// SIMATIC STEP 7 (V5.x) project COB2-CORDNT_040112_LATST
// CPU: CPU 315-2 DP
// station: Hardware
// station: SIMATIC 300(1)
// station: P_ADR_BUS
// program: S7 Program(1)

SYMBOL_TABLE
"DB:RxDTFrmPushCurrent"	DB 15	DB 15	// Pusher Current Data
"DB:RxDTFrmLavelleCurrent"	DB 16	DB 16
"DB: RxEDFrmCharger"	DB 17	DB 17
"DB: RxEDFrmGide"	DB 18	DB 18
"DB: RxEDFrmLoco"	DB 19	DB 19
"DB: RxEDFrmPusher"	DB 20	DB 20
"DB:TxDTFrmCo-Ordination"	DB 21	DB 21
"Level#1<< ---->>Level#2"	DB 23	DB 23
"DB:Data_ReciveBuffer"	DB 29	DB 29
"DB: AutoSPOT"	DB 31	DB 31
"DB: RFModem Freq"	DB 32	DB 32
"DB:HMI TagList"	DB 35	DB 35
"DB:User"	DB 36	DB 36
"DB:InitializationRxBuffe"	DB 39	DB 39
"DB:SndWork DB RS232C"	DB 40	DB 40	// Work DB for P_SND_RK
"DB:RevWork DB RS232C"	DB 41	DB 41	// Work DB for P_RCV_RK
"testng_4_ram_curent_fc45"	DB 45	DB 45	// testng_4_ram_curent_fc45
"FOR_FC-45-OFFLINE"	DB 46	DB 46	// FOR_FC-45-OFFLINE
"IDB_RS232_RM_ChgFreq_SND"	DB 50	FB 8
"IDB_RS232_RM_ChgFreq_RCV"	DB 51	FB 7
"IDB_RS485_AutoSPOT_RCV"	DB 80	FB 7
"DB:USE"	DB 100	DB 100
"P_RCV_ASCII"	FB 7	FB 7	// Receive Data / Provide Data
"P_SND_ASCII"	FB 8	FB 8	// Send Data / Fetch Data
"FC:RF CommunicaTion"	FC 14	FC 14	// RF--Communication & Data Handaling
"FC:OvenIdentification"	FC 19	FC 19
"FC:RxTeleGrm Alocation"	FC 20	FC 20
"FC:RFSndTGram"	FC 21	FC 21	// RF Telegram Sanding
"FC:TxSandTrigger"	FC 23	FC 23
"FC:Co-Ordination Process"	FC 24	FC 24
"FC:SCH_HandLing"	FC 25	FC 25
"FC:CoPLC-------->HMI"	FC 26	FC 26
"FC:FreqChanging"	FC 28	FC 28
"FC:RS232C RCV BLOCK"	FC 29	FC 29
"FC:RS232C SND BLOCK"	FC 30	FC 30	// Communications
"FC: RdAutoSPOT"	FC 31	FC 31	// Oven Identification
"FC:Group_Change_Info"	FC 40	FC 40
"FC_45_OFFLINE"	FC 45	FC 45	// FC_45_OFFLINE
"LoG_0"	M 0.0	BOOL	// LOG 0 BIT
"LoG_1"	M 0.1	BOOL	// LOG 1 BIT
"SysClk_1Sec"	M 1.5	BOOL
"SysClk_2Sec"	M 1.7	BOOL
"CYCL_EXC"	OB 1	OB 1	// Cycle Execution
"PROG_ERR"	OB 121	OB 121	// Programming Error
"MOD_ERR"	OB 122	OB 122	// Module Access Error
"RDREC"	SFB 52	SFB 52	// Read a Process Data Record
"WRREC"	SFB 53	SFB 53	// Write a Process Data Record
"BLKMOV"	SFC 20	SFC 20	// Copy Variables
"FILL"	SFC 21	SFC 21	// Initialize a Memory Area
"VAT_1"	VAT 1	
"ram current testing"	VAT 2		// ram current testing
"all car pos"	VAT 3		// all car pos
"VAT_4"	VAT 4	
"vat5_for_schedule_chek"	VAT 5		// vat5_for_schedule_chek
END_SYMBOL_TABLE

// FB 7: know-how protected block, not included

// FB 8: know-how protected block, not included

FUNCTION "FC:RF CommunicaTion" : VOID	// FC 14
VERSION : 0.1
BEGIN
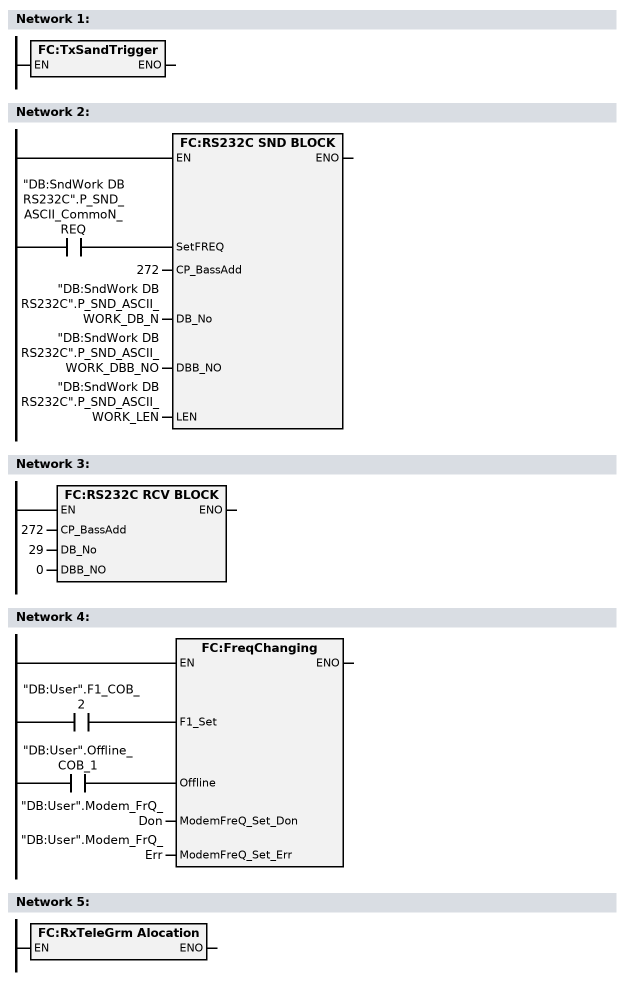
NETWORK
TITLE =
      CALL  "FC:TxSandTrigger";
      NOP   0;
NETWORK
TITLE =
//Data Sand Function Of Radio Modem
      A     "DB:SndWork DB RS232C".P_SND_ASCII_CommoN_REQ;
      =     L 0.0;
      BLD   103;
      CALL  "FC:RS232C SND BLOCK" (
           SetFREQ                  := L 0.0,
           CP_BassAdd               := 272,
           DB_No                    := "DB:SndWork DB RS232C".P_SND_ASCII_WORK_DB_N,
           DBB_NO                   := "DB:SndWork DB RS232C".P_SND_ASCII_WORK_DBB_NO,
           LEN                      := "DB:SndWork DB RS232C".P_SND_ASCII_WORK_LEN);
      NOP   0;
NETWORK
TITLE =
//Data Recive Function Of Radio Modem
      CALL  "FC:RS232C RCV BLOCK" (
           CP_BassAdd               := 272,
           DB_No                    := 29,
           DBB_NO                   := 0);
      NOP   0;
NETWORK
TITLE =
//RF-- Frequency Set In Co-Ordination PLc
      A     "DB:User".F1_COB_2;
      =     L 0.0;
      BLD   103;
      A     "DB:User".Offline_COB_1;
      =     L 0.1;
      BLD   103;
      CALL  "FC:FreqChanging" (
           F1_Set                   := L 0.0,
           Offline                  := L 0.1,
           ModemFreQ_Set_Don        := "DB:User".Modem_FrQ_Don,
           ModemFreQ_Set_Err        := "DB:User".Modem_FrQ_Err);
      NOP   0;
NETWORK
TITLE =
      CALL  "FC:RxTeleGrm Alocation";
      NOP   0;
END_FUNCTION

FUNCTION "FC:OvenIdentification" : VOID	// FC 19
AUTHOR : SKD
NAME : CDSPL
VERSION : 0.1
BEGIN
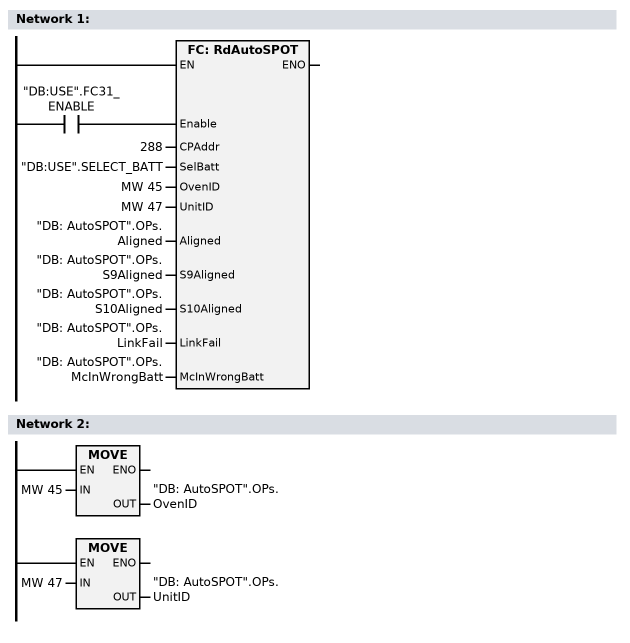
NETWORK
TITLE =
      A     "DB:USE".FC31_ENABLE;
      =     L 0.0;
      BLD   103;
      CALL  "FC: RdAutoSPOT" (
           Enable                   := L 0.0,
           CPAddr                   := 288,
           SelBatt                  := "DB:USE".SELECT_BATT,
           OvenID                   := MW 45,
           UnitID                   := MW 47,
           Aligned                  := "DB: AutoSPOT".OPs.Aligned,
           S9Aligned                := "DB: AutoSPOT".OPs.S9Aligned,
           S10Aligned               := "DB: AutoSPOT".OPs.S10Aligned,
           LinkFail                 := "DB: AutoSPOT".OPs.LinkFail,
           McInWrongBatt            := "DB: AutoSPOT".OPs.McInWrongBatt);
      NOP   0;
NETWORK
TITLE =
      L     MW 45;
      T     "DB: AutoSPOT".OPs.OvenID;
//..
      L     MW 47;
      T     "DB: AutoSPOT".OPs.UnitID;
END_FUNCTION

FUNCTION "FC:RxTeleGrm Alocation" : VOID	// FC 20
VERSION : 0.1
BEGIN
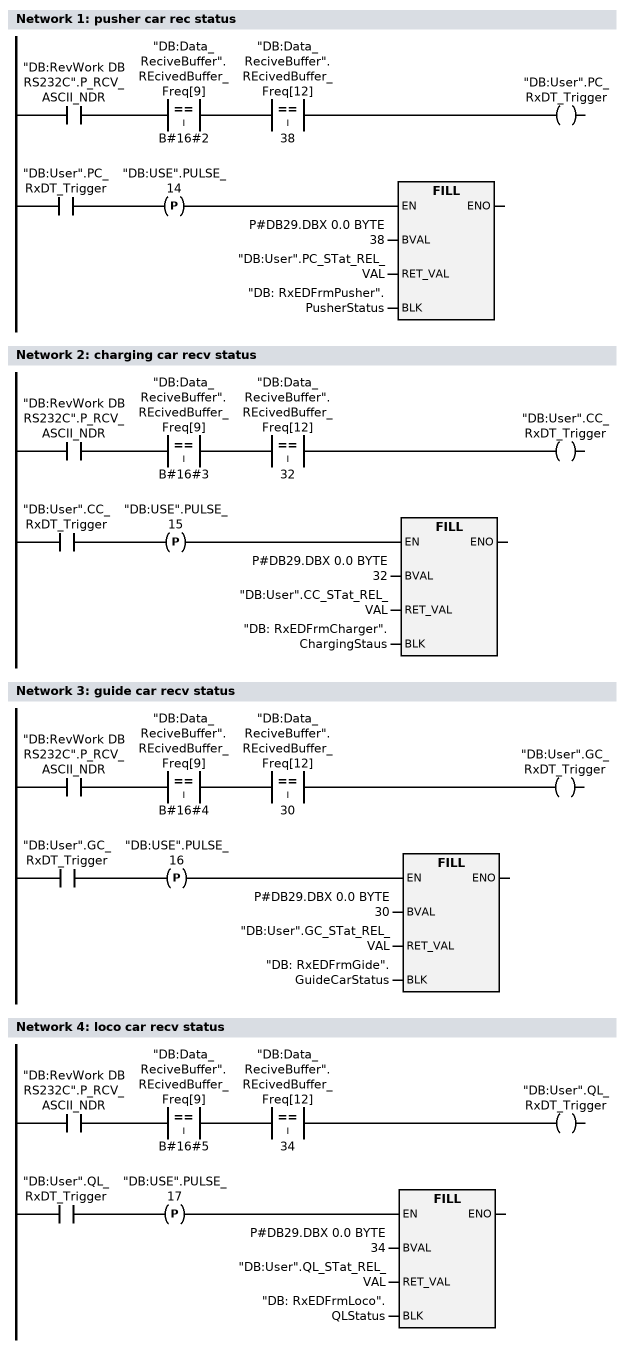
NETWORK
TITLE = pusher car rec status
//pusher car rec status
      A     "DB:RevWork DB RS232C".P_RCV_ASCII_NDR;
      A(;
      L     "DB:Data_ReciveBuffer".REcivedBuffer_Freq[9];
      L     B#16#2;
      ==I;
      );
      A(;
      L     "DB:Data_ReciveBuffer".REcivedBuffer_Freq[12];
      L     38;	//Massege ID
      ==I;
      );
      =     "DB:User".PC_RxDT_Trigger;
//..
      A     "DB:User".PC_RxDT_Trigger;
      FP    "DB:USE".PULSE_14;
      JNB   PC00;
      CALL  "FILL" (
           BVAL                     := P#DB29.DBX 0.0 BYTE 38,
           RET_VAL                  := "DB:User".PC_STat_REL_VAL,
           BLK                      := "DB: RxEDFrmPusher".PusherStatus);
PC00: NOP   0;
NETWORK
TITLE = charging car recv status
//charging car recv status
      A     "DB:RevWork DB RS232C".P_RCV_ASCII_NDR;
      A(;
      L     "DB:Data_ReciveBuffer".REcivedBuffer_Freq[9];
      L     B#16#3;
      ==I;
      );
      A(;
      L     "DB:Data_ReciveBuffer".REcivedBuffer_Freq[12];
      L     32;	//Massege ID
      ==I;
      );
      =     "DB:User".CC_RxDT_Trigger;
//..
      A     "DB:User".CC_RxDT_Trigger;
      FP    "DB:USE".PULSE_15;
      JNB   CC00;
      CALL  "FILL" (
           BVAL                     := P#DB29.DBX 0.0 BYTE 32,
           RET_VAL                  := "DB:User".CC_STat_REL_VAL,
           BLK                      := "DB: RxEDFrmCharger".ChargingStaus);
CC00: NOP   0;
NETWORK
TITLE = guide car recv status
//guide car recv status
      A     "DB:RevWork DB RS232C".P_RCV_ASCII_NDR;
      A(;
      L     "DB:Data_ReciveBuffer".REcivedBuffer_Freq[9];
      L     B#16#4;
      ==I;
      );
      A(;
      L     "DB:Data_ReciveBuffer".REcivedBuffer_Freq[12];
      L     30;	//Massege ID
      ==I;
      );
      =     "DB:User".GC_RxDT_Trigger;
//..
      A     "DB:User".GC_RxDT_Trigger;
      FP    "DB:USE".PULSE_16;
      JNB   GC00;
      CALL  "FILL" (
           BVAL                     := P#DB29.DBX 0.0 BYTE 30,
           RET_VAL                  := "DB:User".GC_STat_REL_VAL,
           BLK                      := "DB: RxEDFrmGide".GuideCarStatus);
GC00: NOP   0;
NETWORK
TITLE = loco car recv status
//Quenching Car Status
      A     "DB:RevWork DB RS232C".P_RCV_ASCII_NDR;
      A(;
      L     "DB:Data_ReciveBuffer".REcivedBuffer_Freq[9];
      L     B#16#5;
      ==I;
      );
      A(;
      L     "DB:Data_ReciveBuffer".REcivedBuffer_Freq[12];
      L     34;	//Massege ID
      ==I;
      );
      =     "DB:User".QL_RxDT_Trigger;
//..
      A     "DB:User".QL_RxDT_Trigger;
      FP    "DB:USE".PULSE_17;
      JNB   QL00;
      CALL  "FILL" (
           BVAL                     := P#DB29.DBX 0.0 BYTE 34,
           RET_VAL                  := "DB:User".QL_STat_REL_VAL,
           BLK                      := "DB: RxEDFrmLoco".QLStatus);
QL00: NOP   0;
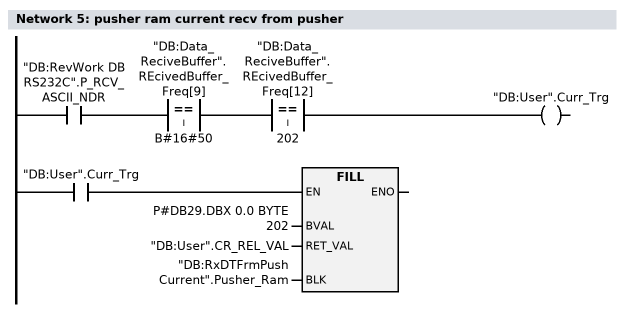
NETWORK
TITLE = pusher ram current recv from pusher
//pusher ram current recv from pusher
      A     "DB:RevWork DB RS232C".P_RCV_ASCII_NDR;
      A(;
      L     "DB:Data_ReciveBuffer".REcivedBuffer_Freq[9];
      L     B#16#50;
      ==I;
      );
      A(;
      L     "DB:Data_ReciveBuffer".REcivedBuffer_Freq[12];
      L     202;	//Massege ID
      ==I;
      );
      =     "DB:User".Curr_Trg;
//..
      A     "DB:User".Curr_Trg;
      JNB   CR00;
      CALL  "FILL" (
           BVAL                     := P#DB29.DBX 0.0 BYTE 202,
           RET_VAL                  := "DB:User".CR_REL_VAL,
           BLK                      := "DB:RxDTFrmPushCurrent".Pusher_Ram);
CR00: NOP   0;
END_FUNCTION

FUNCTION "FC:RFSndTGram" : VOID	// FC 21
VERSION : 0.1
BEGIN
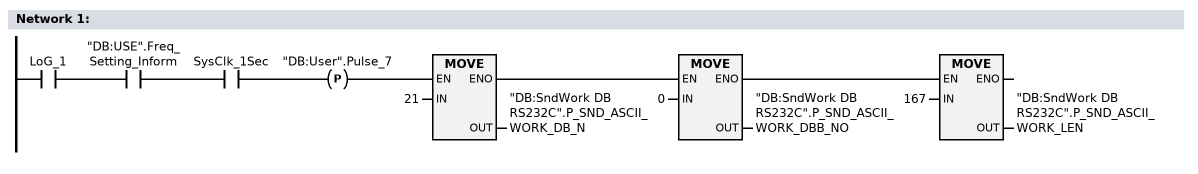
NETWORK
TITLE =
      A(;
      A(;
      A     "LoG_1";
      A     "DB:USE".Freq_Setting_Inform;
      A     "SysClk_1Sec";
      FP    "DB:User".Pulse_7;
      JNB   _001;
      L     21;
      T     "DB:SndWork DB RS232C".P_SND_ASCII_WORK_DB_N;
      SET;
      SAVE;
      CLR;
_001: A     BR;
      );
      JNB   _002;
      L     0;
      T     "DB:SndWork DB RS232C".P_SND_ASCII_WORK_DBB_NO;
      SET;
      SAVE;
      CLR;
_002: A     BR;
      );
      JNB   _003;
      L     167;
      T     "DB:SndWork DB RS232C".P_SND_ASCII_WORK_LEN;
_003: NOP   0;
END_FUNCTION

FUNCTION "FC:TxSandTrigger" : VOID	// FC 23
VERSION : 0.1
BEGIN
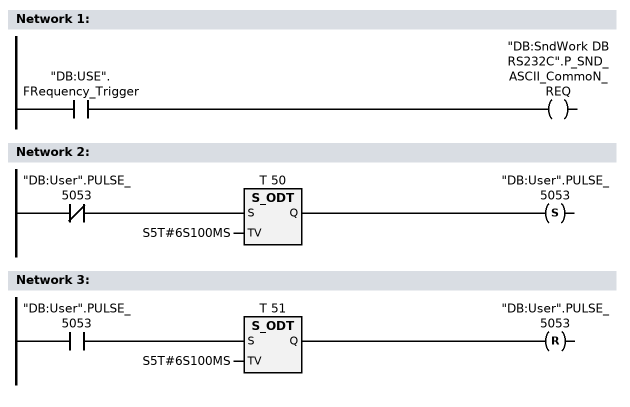
NETWORK
TITLE =
//Machine Grouping and Frequency Setting Triger....for Charging car
      A     "DB:USE".FRequency_Trigger;
      =     "DB:SndWork DB RS232C".P_SND_ASCII_CommoN_REQ;
NETWORK
TITLE =
      AN    "DB:User".PULSE_5053;
      L     S5T#6S100MS;
      SD    T 50;
      NOP   0;
      NOP   0;
      NOP   0;
      A     T 50;
      S     "DB:User".PULSE_5053;
NETWORK
TITLE =
      A     "DB:User".PULSE_5053;
      L     S5T#6S100MS;
      SD    T 51;
      NOP   0;
      NOP   0;
      NOP   0;
      A     T 51;
      R     "DB:User".PULSE_5053;
END_FUNCTION

FUNCTION "FC:Co-Ordination Process" : VOID	// FC 24
VERSION : 0.1
BEGIN
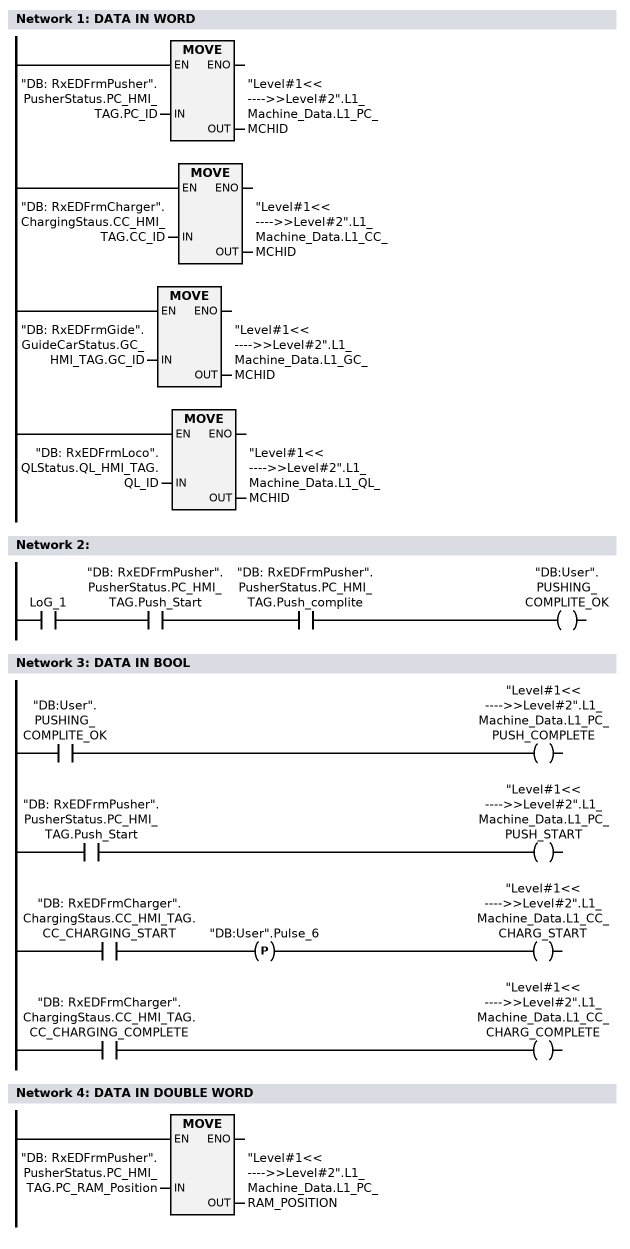
NETWORK
TITLE = DATA IN WORD
      L     "DB: RxEDFrmPusher".PusherStatus.PC_HMI_TAG.PC_ID;
      T     "Level#1<< ---->>Level#2".L1_Machine_Data.L1_PC_MCHID;
//..
      L     "DB: RxEDFrmCharger".ChargingStaus.CC_HMI_TAG.CC_ID;
      T     "Level#1<< ---->>Level#2".L1_Machine_Data.L1_CC_MCHID;
//..
      L     "DB: RxEDFrmGide".GuideCarStatus.GC_HMI_TAG.GC_ID;
      T     "Level#1<< ---->>Level#2".L1_Machine_Data.L1_GC_MCHID;
//..
      L     "DB: RxEDFrmLoco".QLStatus.QL_HMI_TAG.QL_ID;
      T     "Level#1<< ---->>Level#2".L1_Machine_Data.L1_QL_MCHID;
//...
NETWORK
TITLE =
      A     "LoG_1";
      A     "DB: RxEDFrmPusher".PusherStatus.PC_HMI_TAG.Push_Start;
      A     "DB: RxEDFrmPusher".PusherStatus.PC_HMI_TAG.Push_complite;
      =     "DB:User".PUSHING_COMPLITE_OK;
NETWORK
TITLE = DATA IN BOOL
      A     "DB:User".PUSHING_COMPLITE_OK;
      =     "Level#1<< ---->>Level#2".L1_Machine_Data.L1_PC_PUSH_COMPLETE;
//..
      A     "DB: RxEDFrmPusher".PusherStatus.PC_HMI_TAG.Push_Start;
      =     "Level#1<< ---->>Level#2".L1_Machine_Data.L1_PC_PUSH_START;
//..        
      A     "DB: RxEDFrmCharger".ChargingStaus.CC_HMI_TAG.CC_CHARGING_START;
      FP    "DB:User".Pulse_6;
      =     "Level#1<< ---->>Level#2".L1_Machine_Data.L1_CC_CHARG_START;
//..
      A     "DB: RxEDFrmCharger".ChargingStaus.CC_HMI_TAG.CC_CHARGING_COMPLETE;
      =     "Level#1<< ---->>Level#2".L1_Machine_Data.L1_CC_CHARG_COMPLETE;
NETWORK
TITLE = DATA IN DOUBLE WORD
      L     "DB: RxEDFrmPusher".PusherStatus.PC_HMI_TAG.PC_RAM_Position;
      T     "Level#1<< ---->>Level#2".L1_Machine_Data.L1_PC_RAM_POSITION;
//..
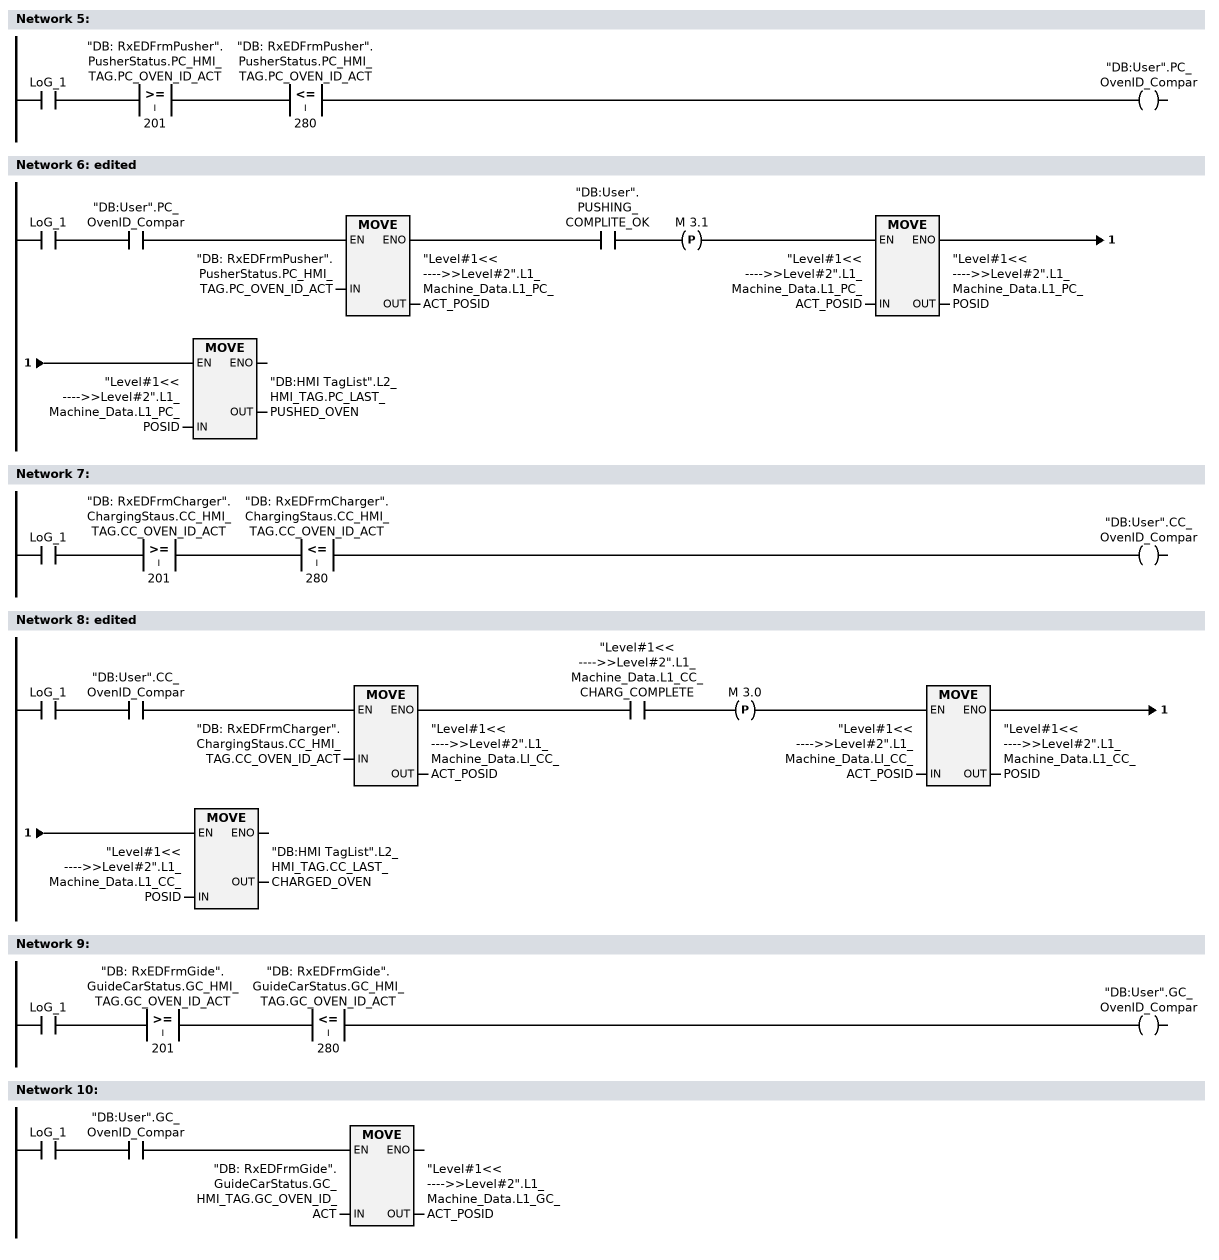
NETWORK
TITLE =
      A     "LoG_1";
      A(;
      L     "DB: RxEDFrmPusher".PusherStatus.PC_HMI_TAG.PC_OVEN_ID_ACT;
      L     201;
      >=I;
      );
      A(;
      L     "DB: RxEDFrmPusher".PusherStatus.PC_HMI_TAG.PC_OVEN_ID_ACT;
      L     280;
      <=I;
      );
      =     "DB:User".PC_OvenID_Compar;
NETWORK
TITLE = edited
//edited last 3  element in this n/w 8 & 6 by me for PC
      A(;
      A(;
      A     "LoG_1";
      A     "DB:User".PC_OvenID_Compar;
      JNB   _001;
      L     "DB: RxEDFrmPusher".PusherStatus.PC_HMI_TAG.PC_OVEN_ID_ACT;
      T     "Level#1<< ---->>Level#2".L1_Machine_Data.L1_PC_ACT_POSID;
      SET;
      SAVE;
      CLR;
_001: A     BR;
      );
      A     "DB:User".PUSHING_COMPLITE_OK;
      FP    M 3.1;
      JNB   _002;
      L     "Level#1<< ---->>Level#2".L1_Machine_Data.L1_PC_ACT_POSID;
      T     "Level#1<< ---->>Level#2".L1_Machine_Data.L1_PC_POSID;
      SET;
      SAVE;
      CLR;
_002: A     BR;
      );
      JNB   _003;
      L     "Level#1<< ---->>Level#2".L1_Machine_Data.L1_PC_POSID;
      T     "DB:HMI TagList".L2_HMI_TAG.PC_LAST_PUSHED_OVEN;
_003: NOP   0;
NETWORK
TITLE =
      A     "LoG_1";
      A(;
      L     "DB: RxEDFrmCharger".ChargingStaus.CC_HMI_TAG.CC_OVEN_ID_ACT;
      L     201;
      >=I;
      );
      A(;
      L     "DB: RxEDFrmCharger".ChargingStaus.CC_HMI_TAG.CC_OVEN_ID_ACT;
      L     280;
      <=I;
      );
      =     "DB:User".CC_OvenID_Compar;
NETWORK
TITLE = edited
//edited last 3  element in this n/w 8 & 6 by me for CC
      A(;
      A(;
      A     "LoG_1";
      A     "DB:User".CC_OvenID_Compar;
      JNB   _004;
      L     "DB: RxEDFrmCharger".ChargingStaus.CC_HMI_TAG.CC_OVEN_ID_ACT;
      T     "Level#1<< ---->>Level#2".L1_Machine_Data.LI_CC_ACT_POSID;
      SET;
      SAVE;
      CLR;
_004: A     BR;
      );
      A     "Level#1<< ---->>Level#2".L1_Machine_Data.L1_CC_CHARG_COMPLETE;
      FP    M 3.0;
      JNB   _005;
      L     "Level#1<< ---->>Level#2".L1_Machine_Data.LI_CC_ACT_POSID;
      T     "Level#1<< ---->>Level#2".L1_Machine_Data.L1_CC_POSID;
      SET;
      SAVE;
      CLR;
_005: A     BR;
      );
      JNB   _006;
      L     "Level#1<< ---->>Level#2".L1_Machine_Data.L1_CC_POSID;
      T     "DB:HMI TagList".L2_HMI_TAG.CC_LAST_CHARGED_OVEN;
_006: NOP   0;
NETWORK
TITLE =
      A     "LoG_1";
      A(;
      L     "DB: RxEDFrmGide".GuideCarStatus.GC_HMI_TAG.GC_OVEN_ID_ACT;
      L     201;
      >=I;
      );
      A(;
      L     "DB: RxEDFrmGide".GuideCarStatus.GC_HMI_TAG.GC_OVEN_ID_ACT;
      L     280;
      <=I;
      );
      =     "DB:User".GC_OvenID_Compar;
NETWORK
TITLE =
      A     "LoG_1";
      A     "DB:User".GC_OvenID_Compar;
      JNB   _007;
      L     "DB: RxEDFrmGide".GuideCarStatus.GC_HMI_TAG.GC_OVEN_ID_ACT;
      T     "Level#1<< ---->>Level#2".L1_Machine_Data.L1_GC_ACT_POSID;
_007: NOP   0;
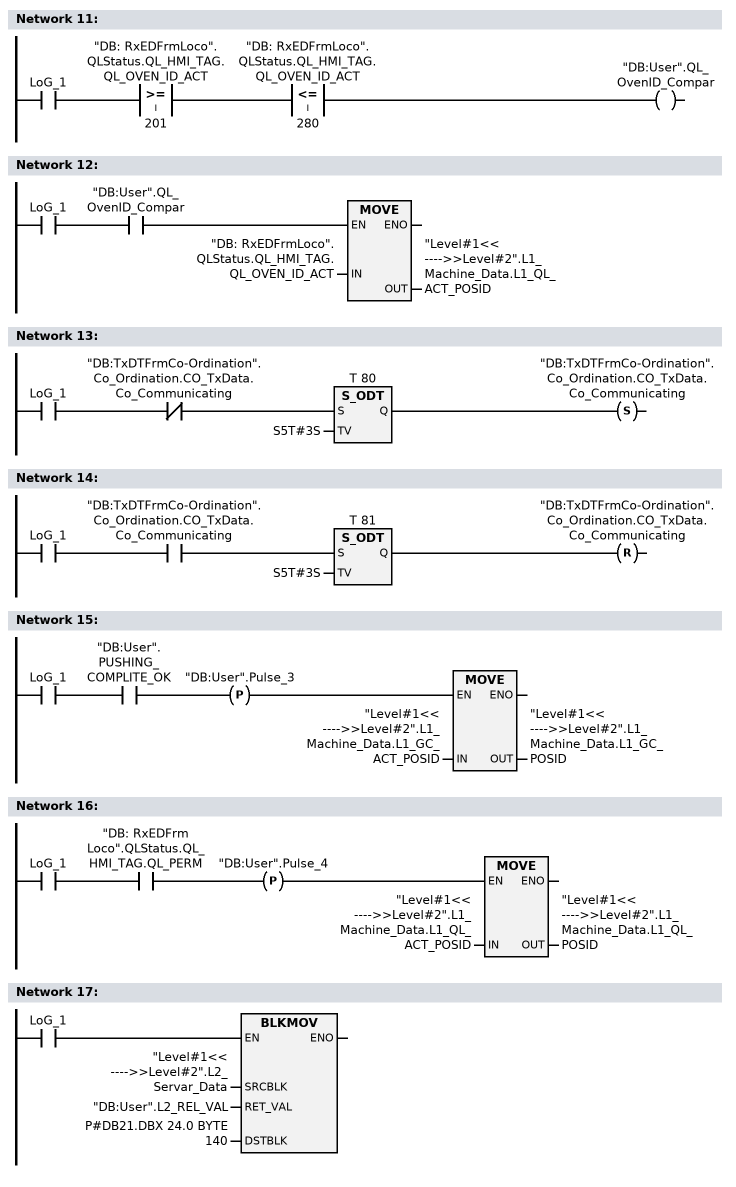
NETWORK
TITLE =
      A     "LoG_1";
      A(;
      L     "DB: RxEDFrmLoco".QLStatus.QL_HMI_TAG.QL_OVEN_ID_ACT;
      L     201;
      >=I;
      );
      A(;
      L     "DB: RxEDFrmLoco".QLStatus.QL_HMI_TAG.QL_OVEN_ID_ACT;
      L     280;
      <=I;
      );
      =     "DB:User".QL_OvenID_Compar;
NETWORK
TITLE =
      A     "LoG_1";
      A     "DB:User".QL_OvenID_Compar;
      JNB   _008;
      L     "DB: RxEDFrmLoco".QLStatus.QL_HMI_TAG.QL_OVEN_ID_ACT;
      T     "Level#1<< ---->>Level#2".L1_Machine_Data.L1_QL_ACT_POSID;
_008: NOP   0;
NETWORK
TITLE =
      A     "LoG_1";
      AN    "DB:TxDTFrmCo-Ordination".Co_Ordination.CO_TxData.Co_Communicating;
      L     S5T#3S;
      SD    T 80;
      NOP   0;
      NOP   0;
      NOP   0;
      A     T 80;
      S     "DB:TxDTFrmCo-Ordination".Co_Ordination.CO_TxData.Co_Communicating;
NETWORK
TITLE =
      A     "LoG_1";
      A     "DB:TxDTFrmCo-Ordination".Co_Ordination.CO_TxData.Co_Communicating;
      L     S5T#3S;
      SD    T 81;
      NOP   0;
      NOP   0;
      NOP   0;
      A     T 81;
      R     "DB:TxDTFrmCo-Ordination".Co_Ordination.CO_TxData.Co_Communicating;
NETWORK
TITLE =
      A     "LoG_1";
      A     "DB:User".PUSHING_COMPLITE_OK;
      FP    "DB:User".Pulse_3;
      JNB   _009;
      L     "Level#1<< ---->>Level#2".L1_Machine_Data.L1_GC_ACT_POSID;
      T     "Level#1<< ---->>Level#2".L1_Machine_Data.L1_GC_POSID;
_009: NOP   0;
NETWORK
TITLE =
      A     "LoG_1";
      A     "DB: RxEDFrmLoco".QLStatus.QL_HMI_TAG.QL_PERM;
      FP    "DB:User".Pulse_4;
      JNB   _00a;
      L     "Level#1<< ---->>Level#2".L1_Machine_Data.L1_QL_ACT_POSID;
      T     "Level#1<< ---->>Level#2".L1_Machine_Data.L1_QL_POSID;
_00a: NOP   0;
NETWORK
TITLE =
      A     "LoG_1";
      JNB   _00b;
      CALL  "BLKMOV" (
           SRCBLK                   := "Level#1<< ---->>Level#2".L2_Servar_Data,
           RET_VAL                  := "DB:User".L2_REL_VAL,
           DSTBLK                   := P#DB21.DBX 24.0 BYTE 140);
_00b: NOP   0;
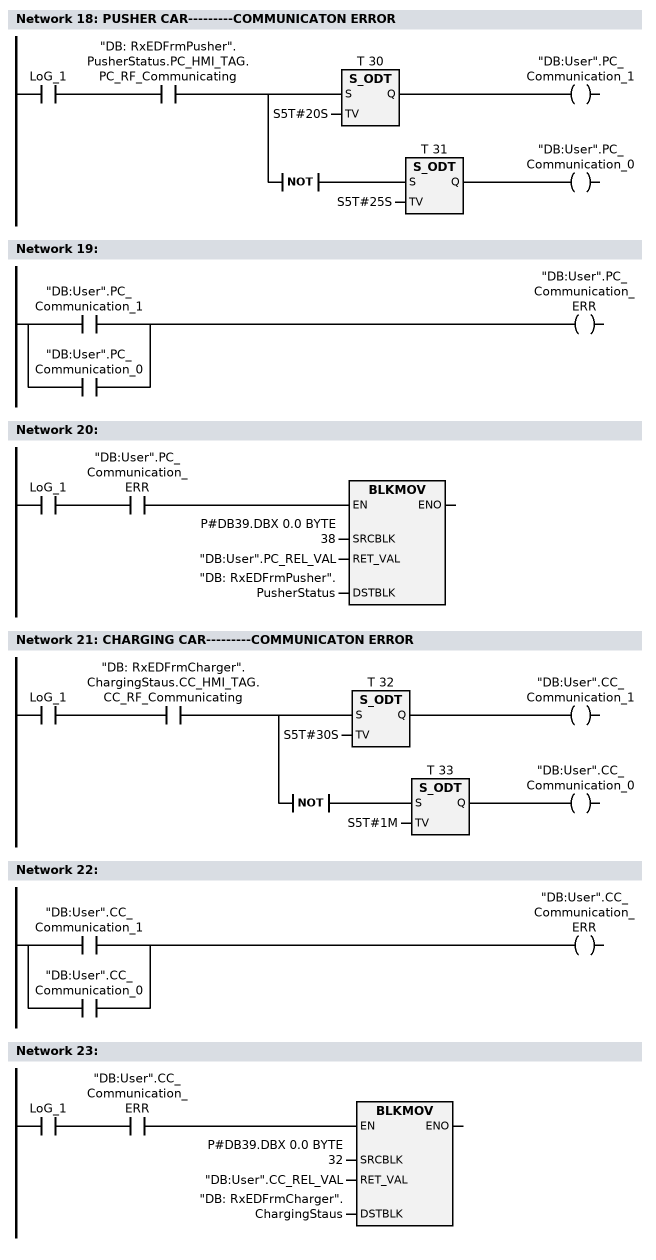
NETWORK
TITLE = PUSHER CAR---------COMMUNICATON ERROR
      A     "LoG_1";
      A     "DB: RxEDFrmPusher".PusherStatus.PC_HMI_TAG.PC_RF_Communicating;
      =     L 0.0;
      A     L 0.0;
      L     S5T#20S;
      SD    T 30;
      NOP   0;
      NOP   0;
      NOP   0;
      A     T 30;
      =     "DB:User".PC_Communication_1;
      A     L 0.0;
      NOT;
      L     S5T#25S;
      SD    T 31;
      NOP   0;
      NOP   0;
      NOP   0;
      A     T 31;
      =     "DB:User".PC_Communication_0;
NETWORK
TITLE =
//Pusher Car Error Bit
      O     "DB:User".PC_Communication_1;
      O     "DB:User".PC_Communication_0;
      =     "DB:User".PC_Communication_ERR;
NETWORK
TITLE =
//Pusher Car Status Initialisation 
      A     "LoG_1";
      A     "DB:User".PC_Communication_ERR;
      JNB   _00c;
      CALL  "BLKMOV" (
           SRCBLK                   := P#DB39.DBX 0.0 BYTE 38,
           RET_VAL                  := "DB:User".PC_REL_VAL,
           DSTBLK                   := "DB: RxEDFrmPusher".PusherStatus);
_00c: NOP   0;
NETWORK
TITLE = CHARGING CAR---------COMMUNICATON ERROR
      A     "LoG_1";
      A     "DB: RxEDFrmCharger".ChargingStaus.CC_HMI_TAG.CC_RF_Communicating;
      =     L 0.0;
      A     L 0.0;
      L     S5T#30S;
      SD    T 32;
      NOP   0;
      NOP   0;
      NOP   0;
      A     T 32;
      =     "DB:User".CC_Communication_1;
      A     L 0.0;
      NOT;
      L     S5T#1M;
      SD    T 33;
      NOP   0;
      NOP   0;
      NOP   0;
      A     T 33;
      =     "DB:User".CC_Communication_0;
NETWORK
TITLE =
//Charging Car Error Bit
      O     "DB:User".CC_Communication_1;
      O     "DB:User".CC_Communication_0;
      =     "DB:User".CC_Communication_ERR;
NETWORK
TITLE =
// Carging Car Status Initialisation 
      A     "LoG_1";
      A     "DB:User".CC_Communication_ERR;
      JNB   _00d;
      CALL  "BLKMOV" (
           SRCBLK                   := P#DB39.DBX 0.0 BYTE 32,
           RET_VAL                  := "DB:User".CC_REL_VAL,
           DSTBLK                   := "DB: RxEDFrmCharger".ChargingStaus);
_00d: NOP   0;
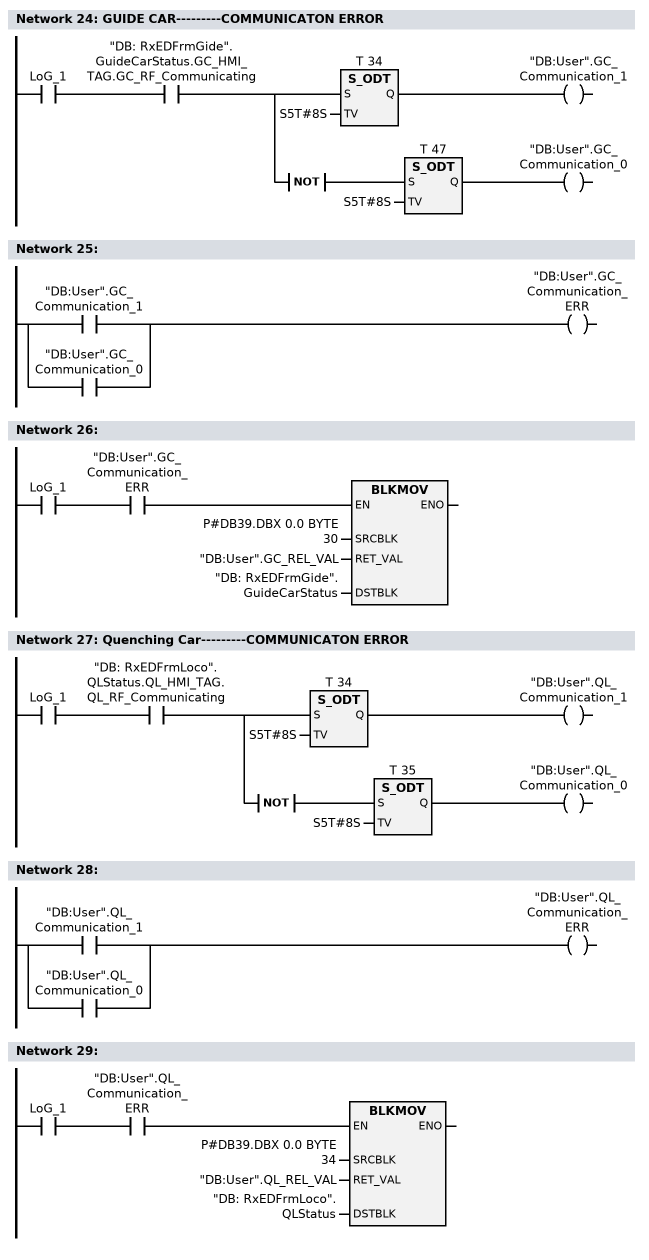
NETWORK
TITLE = GUIDE CAR---------COMMUNICATON ERROR
      A     "LoG_1";
      A     "DB: RxEDFrmGide".GuideCarStatus.GC_HMI_TAG.GC_RF_Communicating;
      =     L 0.0;
      A     L 0.0;
      L     S5T#8S;
      SD    T 34;
      NOP   0;
      NOP   0;
      NOP   0;
      A     T 34;
      =     "DB:User".GC_Communication_1;
      A     L 0.0;
      NOT;
      L     S5T#8S;
      SD    T 47;
      NOP   0;
      NOP   0;
      NOP   0;
      A     T 47;
      =     "DB:User".GC_Communication_0;
NETWORK
TITLE =
//Guide Car Error Bit
      O     "DB:User".GC_Communication_1;
      O     "DB:User".GC_Communication_0;
      =     "DB:User".GC_Communication_ERR;
NETWORK
TITLE =
//Guide Car Status Initialisation 
      A     "LoG_1";
      A     "DB:User".GC_Communication_ERR;
      JNB   _00e;
      CALL  "BLKMOV" (
           SRCBLK                   := P#DB39.DBX 0.0 BYTE 30,
           RET_VAL                  := "DB:User".GC_REL_VAL,
           DSTBLK                   := "DB: RxEDFrmGide".GuideCarStatus);
_00e: NOP   0;
NETWORK
TITLE = Quenching Car---------COMMUNICATON ERROR
      A     "LoG_1";
      A     "DB: RxEDFrmLoco".QLStatus.QL_HMI_TAG.QL_RF_Communicating;
      =     L 0.0;
      A     L 0.0;
      L     S5T#8S;
      SD    T 34;
      NOP   0;
      NOP   0;
      NOP   0;
      A     T 34;
      =     "DB:User".QL_Communication_1;
      A     L 0.0;
      NOT;
      L     S5T#8S;
      SD    T 35;
      NOP   0;
      NOP   0;
      NOP   0;
      A     T 35;
      =     "DB:User".QL_Communication_0;
NETWORK
TITLE =
//Quenching Car Error Bit
      O     "DB:User".QL_Communication_1;
      O     "DB:User".QL_Communication_0;
      =     "DB:User".QL_Communication_ERR;
NETWORK
TITLE =
//Quenching Car Status Initialisation 
      A     "LoG_1";
      A     "DB:User".QL_Communication_ERR;
      JNB   _00f;
      CALL  "BLKMOV" (
           SRCBLK                   := P#DB39.DBX 0.0 BYTE 34,
           RET_VAL                  := "DB:User".QL_REL_VAL,
           DSTBLK                   := "DB: RxEDFrmLoco".QLStatus);
_00f: NOP   0;
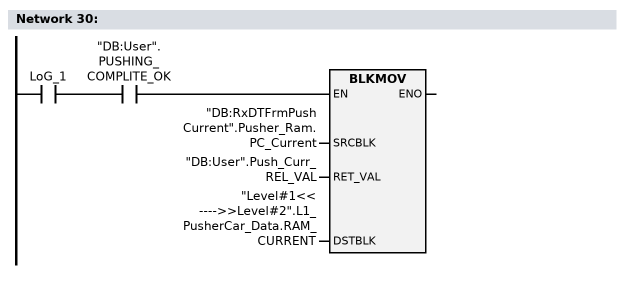
NETWORK
TITLE =
      A     "LoG_1";
      A     "DB:User".PUSHING_COMPLITE_OK;
      JNB   _010;
      CALL  "BLKMOV" (
           SRCBLK                   := "DB:RxDTFrmPushCurrent".Pusher_Ram.PC_Current,
           RET_VAL                  := "DB:User".Push_Curr_REL_VAL,
           DSTBLK                   := "Level#1<< ---->>Level#2".L1_PusherCar_Data.RAM_CURRENT);
_010: NOP   0;
END_FUNCTION

FUNCTION "FC:SCH_HandLing" : VOID	// FC 25
VERSION : 0.1
VAR_TEMP
  Subtract_Valu_1 : INT ;
  Addition_Valu_1 : INT ;
  Subtract_Valu_2 : INT ;
  Addition_Valu_2 : INT ;
  Subtract_Valu_3 : INT ;
  Addition_Valu_3 : INT ;
  Subtract_Valu_4 : INT ;
  Addition_Valu_4 : INT ;
  Subtract_Valu_5 : INT ;
  Addition_Valu_5 : INT ;
END_VAR
BEGIN
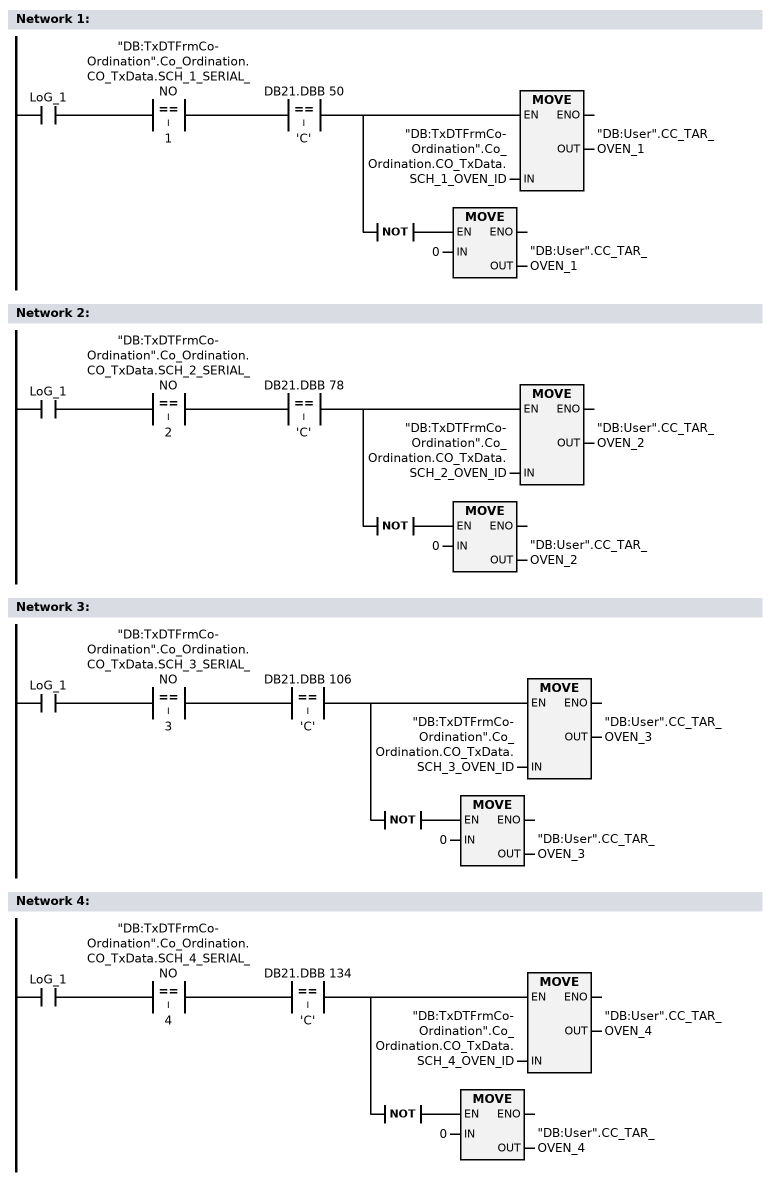
NETWORK
TITLE =
      A     "LoG_1";
      A(;
      L     "DB:TxDTFrmCo-Ordination".Co_Ordination.CO_TxData.SCH_1_SERIAL_NO;
      L     1;
      ==I;
      );
      A(;
      L     DB21.DBB 50;
      L     'C';
      ==I;
      );
      =     L 22.0;
      A     L 22.0;
      JNB   _01E;
      L     "DB:TxDTFrmCo-Ordination".Co_Ordination.CO_TxData.SCH_1_OVEN_ID;
      T     "DB:User".CC_TAR_OVEN_1;
_01E: NOP   0;
      A     L 22.0;
      NOT;
      JNB   _01F;
      L     0;
      T     "DB:User".CC_TAR_OVEN_1;
_01F: NOP   0;
NETWORK
TITLE =
      A     "LoG_1";
      A(;
      L     "DB:TxDTFrmCo-Ordination".Co_Ordination.CO_TxData.SCH_2_SERIAL_NO;
      L     2;
      ==I;
      );
      A(;
      L     DB21.DBB 78;
      L     'C';
      ==I;
      );
      =     L 23.0;
      A     L 23.0;
      JNB   _01e;
      L     "DB:TxDTFrmCo-Ordination".Co_Ordination.CO_TxData.SCH_2_OVEN_ID;
      T     "DB:User".CC_TAR_OVEN_2;
_01e: NOP   0;
      A     L 23.0;
      NOT;
      JNB   _01f;
      L     0;
      T     "DB:User".CC_TAR_OVEN_2;
_01f: NOP   0;
NETWORK
TITLE =
      A     "LoG_1";
      A(;
      L     "DB:TxDTFrmCo-Ordination".Co_Ordination.CO_TxData.SCH_3_SERIAL_NO;
      L     3;
      ==I;
      );
      A(;
      L     DB21.DBB 106;
      L     'C';
      ==I;
      );
      =     L 24.0;
      A     L 24.0;
      JNB   _020;
      L     "DB:TxDTFrmCo-Ordination".Co_Ordination.CO_TxData.SCH_3_OVEN_ID;
      T     "DB:User".CC_TAR_OVEN_3;
_020: NOP   0;
      A     L 24.0;
      NOT;
      JNB   _021;
      L     0;
      T     "DB:User".CC_TAR_OVEN_3;
_021: NOP   0;
NETWORK
TITLE =
      A     "LoG_1";
      A(;
      L     "DB:TxDTFrmCo-Ordination".Co_Ordination.CO_TxData.SCH_4_SERIAL_NO;
      L     4;
      ==I;
      );
      A(;
      L     DB21.DBB 134;
      L     'C';
      ==I;
      );
      =     L 25.0;
      A     L 25.0;
      JNB   _001;
      L     "DB:TxDTFrmCo-Ordination".Co_Ordination.CO_TxData.SCH_4_OVEN_ID;
      T     "DB:User".CC_TAR_OVEN_4;
_001: NOP   0;
      A     L 25.0;
      NOT;
      JNB   _002;
      L     0;
      T     "DB:User".CC_TAR_OVEN_4;
_002: NOP   0;
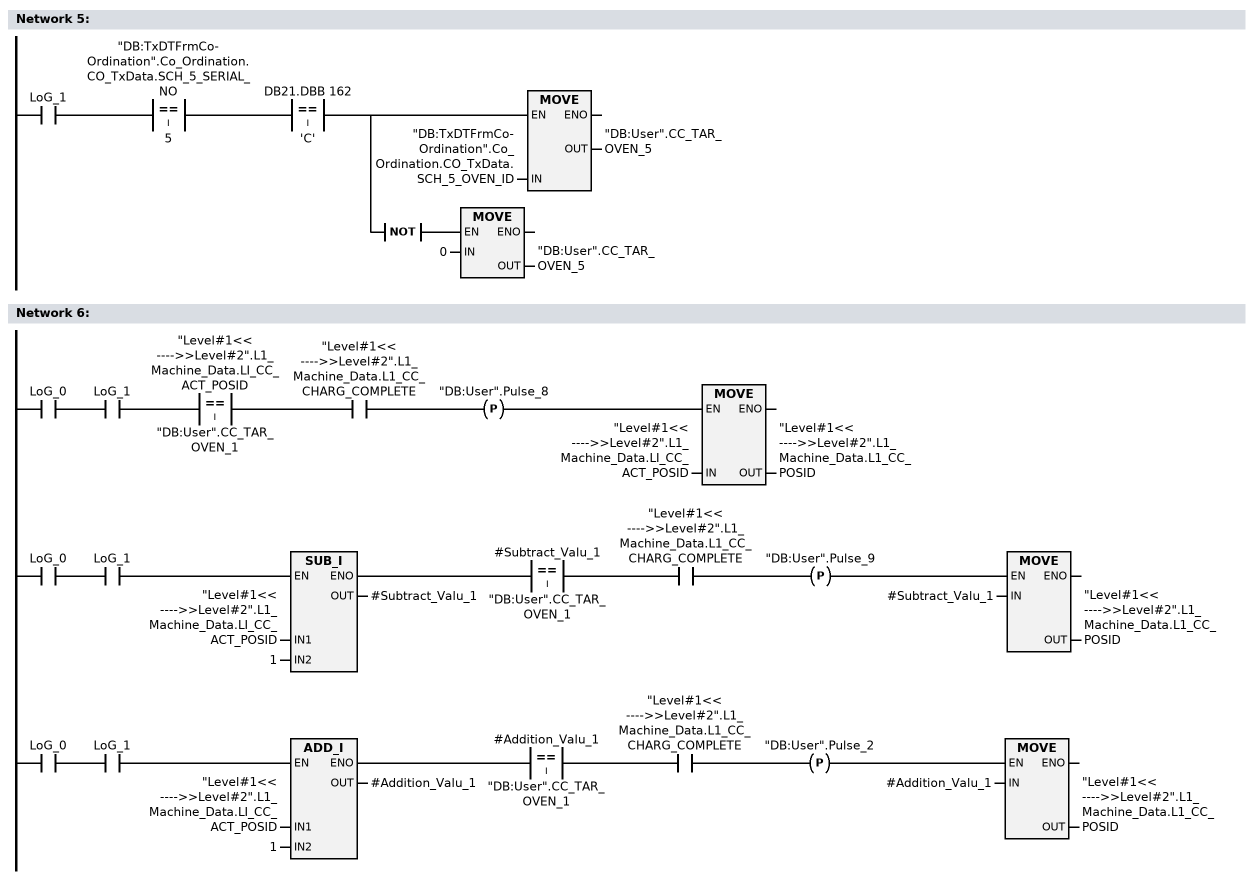
NETWORK
TITLE =
      A     "LoG_1";
      A(;
      L     "DB:TxDTFrmCo-Ordination".Co_Ordination.CO_TxData.SCH_5_SERIAL_NO;
      L     5;
      ==I;
      );
      A(;
      L     DB21.DBB 162;
      L     'C';
      ==I;
      );
      =     L 26.0;
      A     L 26.0;
      JNB   _024;
      L     "DB:TxDTFrmCo-Ordination".Co_Ordination.CO_TxData.SCH_5_OVEN_ID;
      T     "DB:User".CC_TAR_OVEN_5;
_024: NOP   0;
      A     L 26.0;
      NOT;
      JNB   _025;
      L     0;
      T     "DB:User".CC_TAR_OVEN_5;
_025: NOP   0;
NETWORK
TITLE =
      A     "LoG_0";
      A     "LoG_1";
      =     L 30.0;
      A(;
      A     L 30.0;
      JNB   _003;
      L     "Level#1<< ---->>Level#2".L1_Machine_Data.LI_CC_ACT_POSID;
      L     1;
      -I;
      T     #Subtract_Valu_1;
      AN    OV;
      SAVE;
      CLR;
_003: A     BR;
      );
      A(;
      L     #Subtract_Valu_1;
      L     "DB:User".CC_TAR_OVEN_1;
      ==I;
      );
      A     "Level#1<< ---->>Level#2".L1_Machine_Data.L1_CC_CHARG_COMPLETE;
      FP    "DB:User".Pulse_9;
      JNB   _004;
      L     #Subtract_Valu_1;
      T     "Level#1<< ---->>Level#2".L1_Machine_Data.L1_CC_POSID;
_004: NOP   0;
      A(;
      A     L 30.0;
      JNB   _005;
      L     "Level#1<< ---->>Level#2".L1_Machine_Data.LI_CC_ACT_POSID;
      L     1;
      +I;
      T     #Addition_Valu_1;
      AN    OV;
      SAVE;
      CLR;
_005: A     BR;
      );
      A(;
      L     #Addition_Valu_1;
      L     "DB:User".CC_TAR_OVEN_1;
      ==I;
      );
      A     "Level#1<< ---->>Level#2".L1_Machine_Data.L1_CC_CHARG_COMPLETE;
      FP    "DB:User".Pulse_2;
      JNB   _006;
      L     #Addition_Valu_1;
      T     "Level#1<< ---->>Level#2".L1_Machine_Data.L1_CC_POSID;
_006: NOP   0;
      A     L 30.0;
      A(;
      L     "Level#1<< ---->>Level#2".L1_Machine_Data.LI_CC_ACT_POSID;
      L     "DB:User".CC_TAR_OVEN_1;
      ==I;
      );
      A     "Level#1<< ---->>Level#2".L1_Machine_Data.L1_CC_CHARG_COMPLETE;
      FP    "DB:User".Pulse_8;
      JNB   _007;
      L     "Level#1<< ---->>Level#2".L1_Machine_Data.LI_CC_ACT_POSID;
      T     "Level#1<< ---->>Level#2".L1_Machine_Data.L1_CC_POSID;
_007: NOP   0;
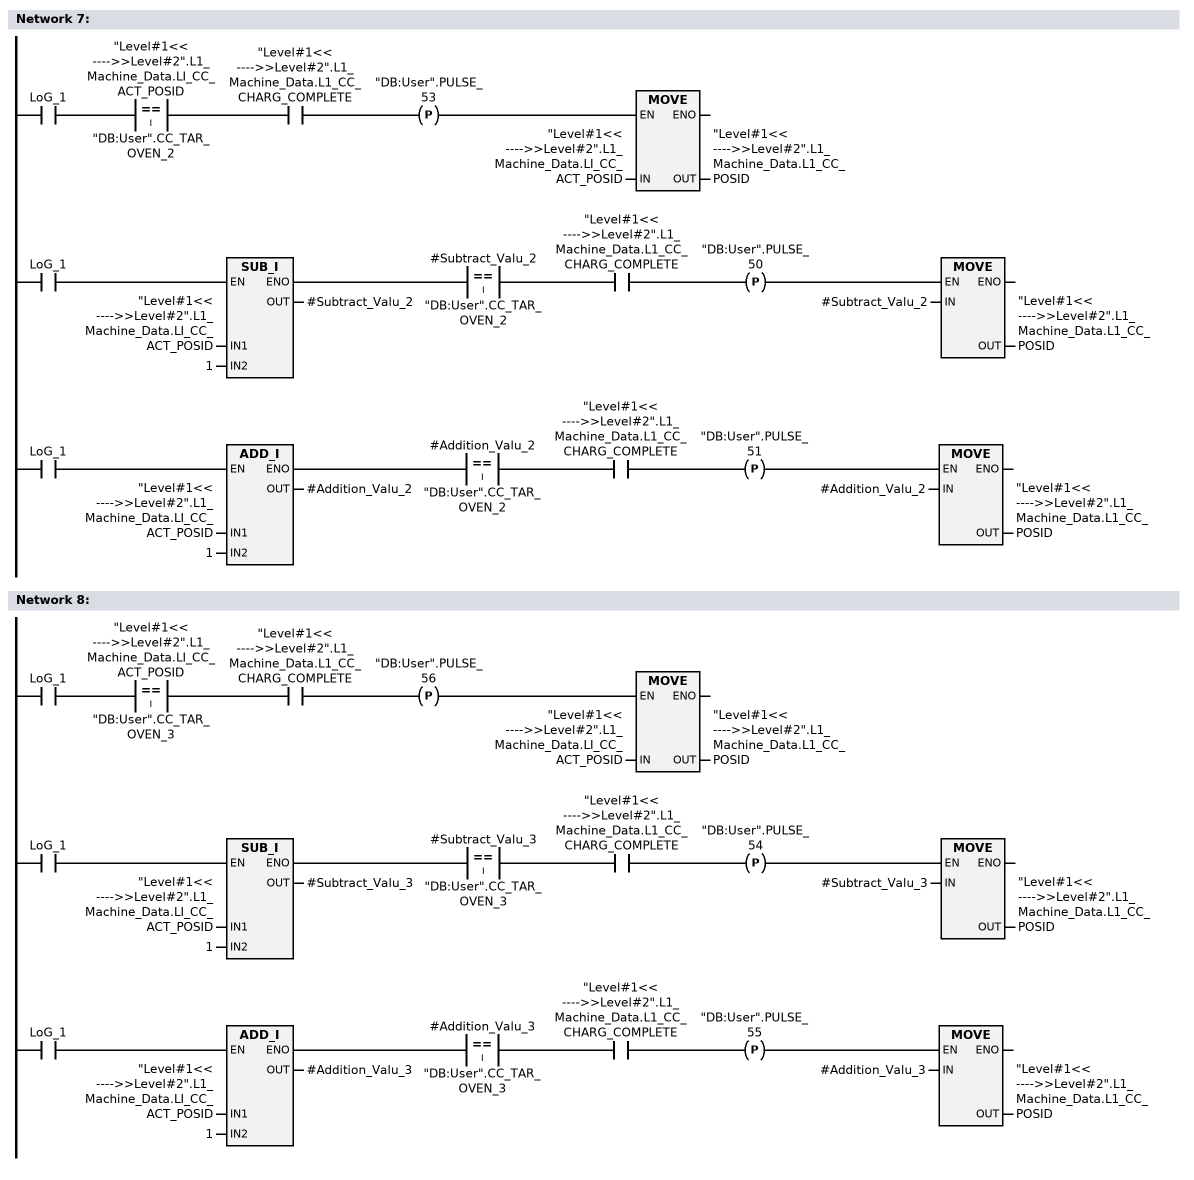
NETWORK
TITLE =
      A     "LoG_1";
      =     L 30.0;
      A(;
      A     L 30.0;
      JNB   _008;
      L     "Level#1<< ---->>Level#2".L1_Machine_Data.LI_CC_ACT_POSID;
      L     1;
      -I;
      T     #Subtract_Valu_2;
      AN    OV;
      SAVE;
      CLR;
_008: A     BR;
      );
      A(;
      L     #Subtract_Valu_2;
      L     "DB:User".CC_TAR_OVEN_2;
      ==I;
      );
      A     "Level#1<< ---->>Level#2".L1_Machine_Data.L1_CC_CHARG_COMPLETE;
      FP    "DB:User".PULSE_50;
      JNB   _009;
      L     #Subtract_Valu_2;
      T     "Level#1<< ---->>Level#2".L1_Machine_Data.L1_CC_POSID;
_009: NOP   0;
      A(;
      A     L 30.0;
      JNB   _00a;
      L     "Level#1<< ---->>Level#2".L1_Machine_Data.LI_CC_ACT_POSID;
      L     1;
      +I;
      T     #Addition_Valu_2;
      AN    OV;
      SAVE;
      CLR;
_00a: A     BR;
      );
      A(;
      L     #Addition_Valu_2;
      L     "DB:User".CC_TAR_OVEN_2;
      ==I;
      );
      A     "Level#1<< ---->>Level#2".L1_Machine_Data.L1_CC_CHARG_COMPLETE;
      FP    "DB:User".PULSE_51;
      JNB   _00b;
      L     #Addition_Valu_2;
      T     "Level#1<< ---->>Level#2".L1_Machine_Data.L1_CC_POSID;
_00b: NOP   0;
      A     L 30.0;
      A(;
      L     "Level#1<< ---->>Level#2".L1_Machine_Data.LI_CC_ACT_POSID;
      L     "DB:User".CC_TAR_OVEN_2;
      ==I;
      );
      A     "Level#1<< ---->>Level#2".L1_Machine_Data.L1_CC_CHARG_COMPLETE;
      FP    "DB:User".PULSE_53;
      JNB   _00c;
      L     "Level#1<< ---->>Level#2".L1_Machine_Data.LI_CC_ACT_POSID;
      T     "Level#1<< ---->>Level#2".L1_Machine_Data.L1_CC_POSID;
_00c: NOP   0;
NETWORK
TITLE =
      A     "LoG_1";
      =     L 30.0;
      A(;
      A     L 30.0;
      JNB   _00d;
      L     "Level#1<< ---->>Level#2".L1_Machine_Data.LI_CC_ACT_POSID;
      L     1;
      -I;
      T     #Subtract_Valu_3;
      AN    OV;
      SAVE;
      CLR;
_00d: A     BR;
      );
      A(;
      L     #Subtract_Valu_3;
      L     "DB:User".CC_TAR_OVEN_3;
      ==I;
      );
      A     "Level#1<< ---->>Level#2".L1_Machine_Data.L1_CC_CHARG_COMPLETE;
      FP    "DB:User".PULSE_54;
      JNB   _00e;
      L     #Subtract_Valu_3;
      T     "Level#1<< ---->>Level#2".L1_Machine_Data.L1_CC_POSID;
_00e: NOP   0;
      A(;
      A     L 30.0;
      JNB   _00f;
      L     "Level#1<< ---->>Level#2".L1_Machine_Data.LI_CC_ACT_POSID;
      L     1;
      +I;
      T     #Addition_Valu_3;
      AN    OV;
      SAVE;
      CLR;
_00f: A     BR;
      );
      A(;
      L     #Addition_Valu_3;
      L     "DB:User".CC_TAR_OVEN_3;
      ==I;
      );
      A     "Level#1<< ---->>Level#2".L1_Machine_Data.L1_CC_CHARG_COMPLETE;
      FP    "DB:User".PULSE_55;
      JNB   _010;
      L     #Addition_Valu_3;
      T     "Level#1<< ---->>Level#2".L1_Machine_Data.L1_CC_POSID;
_010: NOP   0;
      A     L 30.0;
      A(;
      L     "Level#1<< ---->>Level#2".L1_Machine_Data.LI_CC_ACT_POSID;
      L     "DB:User".CC_TAR_OVEN_3;
      ==I;
      );
      A     "Level#1<< ---->>Level#2".L1_Machine_Data.L1_CC_CHARG_COMPLETE;
      FP    "DB:User".PULSE_56;
      JNB   _011;
      L     "Level#1<< ---->>Level#2".L1_Machine_Data.LI_CC_ACT_POSID;
      T     "Level#1<< ---->>Level#2".L1_Machine_Data.L1_CC_POSID;
_011: NOP   0;
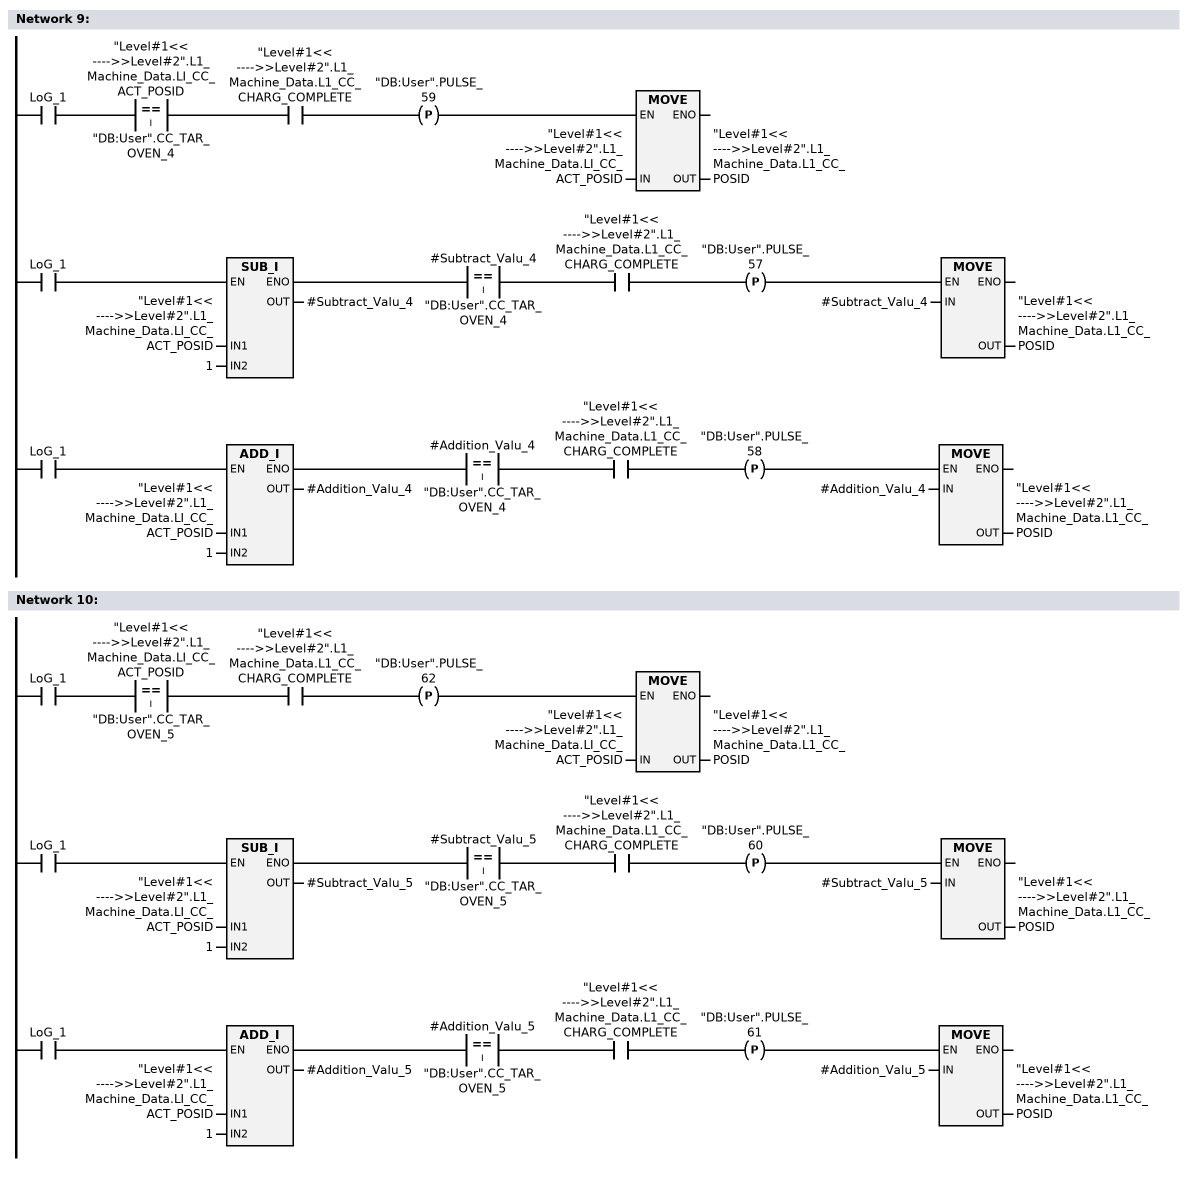
NETWORK
TITLE =
      A     "LoG_1";
      =     L 30.0;
      A(;
      A     L 30.0;
      JNB   _012;
      L     "Level#1<< ---->>Level#2".L1_Machine_Data.LI_CC_ACT_POSID;
      L     1;
      -I;
      T     #Subtract_Valu_4;
      AN    OV;
      SAVE;
      CLR;
_012: A     BR;
      );
      A(;
      L     #Subtract_Valu_4;
      L     "DB:User".CC_TAR_OVEN_4;
      ==I;
      );
      A     "Level#1<< ---->>Level#2".L1_Machine_Data.L1_CC_CHARG_COMPLETE;
      FP    "DB:User".PULSE_57;
      JNB   _013;
      L     #Subtract_Valu_4;
      T     "Level#1<< ---->>Level#2".L1_Machine_Data.L1_CC_POSID;
_013: NOP   0;
      A(;
      A     L 30.0;
      JNB   _014;
      L     "Level#1<< ---->>Level#2".L1_Machine_Data.LI_CC_ACT_POSID;
      L     1;
      +I;
      T     #Addition_Valu_4;
      AN    OV;
      SAVE;
      CLR;
_014: A     BR;
      );
      A(;
      L     #Addition_Valu_4;
      L     "DB:User".CC_TAR_OVEN_4;
      ==I;
      );
      A     "Level#1<< ---->>Level#2".L1_Machine_Data.L1_CC_CHARG_COMPLETE;
      FP    "DB:User".PULSE_58;
      JNB   _015;
      L     #Addition_Valu_4;
      T     "Level#1<< ---->>Level#2".L1_Machine_Data.L1_CC_POSID;
_015: NOP   0;
      A     L 30.0;
      A(;
      L     "Level#1<< ---->>Level#2".L1_Machine_Data.LI_CC_ACT_POSID;
      L     "DB:User".CC_TAR_OVEN_4;
      ==I;
      );
      A     "Level#1<< ---->>Level#2".L1_Machine_Data.L1_CC_CHARG_COMPLETE;
      FP    "DB:User".PULSE_59;
      JNB   _016;
      L     "Level#1<< ---->>Level#2".L1_Machine_Data.LI_CC_ACT_POSID;
      T     "Level#1<< ---->>Level#2".L1_Machine_Data.L1_CC_POSID;
_016: NOP   0;
NETWORK
TITLE =
      A     "LoG_1";
      =     L 30.0;
      A(;
      A     L 30.0;
      JNB   _017;
      L     "Level#1<< ---->>Level#2".L1_Machine_Data.LI_CC_ACT_POSID;
      L     1;
      -I;
      T     #Subtract_Valu_5;
      AN    OV;
      SAVE;
      CLR;
_017: A     BR;
      );
      A(;
      L     #Subtract_Valu_5;
      L     "DB:User".CC_TAR_OVEN_5;
      ==I;
      );
      A     "Level#1<< ---->>Level#2".L1_Machine_Data.L1_CC_CHARG_COMPLETE;
      FP    "DB:User".PULSE_60;
      JNB   _018;
      L     #Subtract_Valu_5;
      T     "Level#1<< ---->>Level#2".L1_Machine_Data.L1_CC_POSID;
_018: NOP   0;
      A(;
      A     L 30.0;
      JNB   _019;
      L     "Level#1<< ---->>Level#2".L1_Machine_Data.LI_CC_ACT_POSID;
      L     1;
      +I;
      T     #Addition_Valu_5;
      AN    OV;
      SAVE;
      CLR;
_019: A     BR;
      );
      A(;
      L     #Addition_Valu_5;
      L     "DB:User".CC_TAR_OVEN_5;
      ==I;
      );
      A     "Level#1<< ---->>Level#2".L1_Machine_Data.L1_CC_CHARG_COMPLETE;
      FP    "DB:User".PULSE_61;
      JNB   _01a;
      L     #Addition_Valu_5;
      T     "Level#1<< ---->>Level#2".L1_Machine_Data.L1_CC_POSID;
_01a: NOP   0;
      A     L 30.0;
      A(;
      L     "Level#1<< ---->>Level#2".L1_Machine_Data.LI_CC_ACT_POSID;
      L     "DB:User".CC_TAR_OVEN_5;
      ==I;
      );
      A     "Level#1<< ---->>Level#2".L1_Machine_Data.L1_CC_CHARG_COMPLETE;
      FP    "DB:User".PULSE_62;
      JNB   _01b;
      L     "Level#1<< ---->>Level#2".L1_Machine_Data.LI_CC_ACT_POSID;
      T     "Level#1<< ---->>Level#2".L1_Machine_Data.L1_CC_POSID;
_01b: NOP   0;
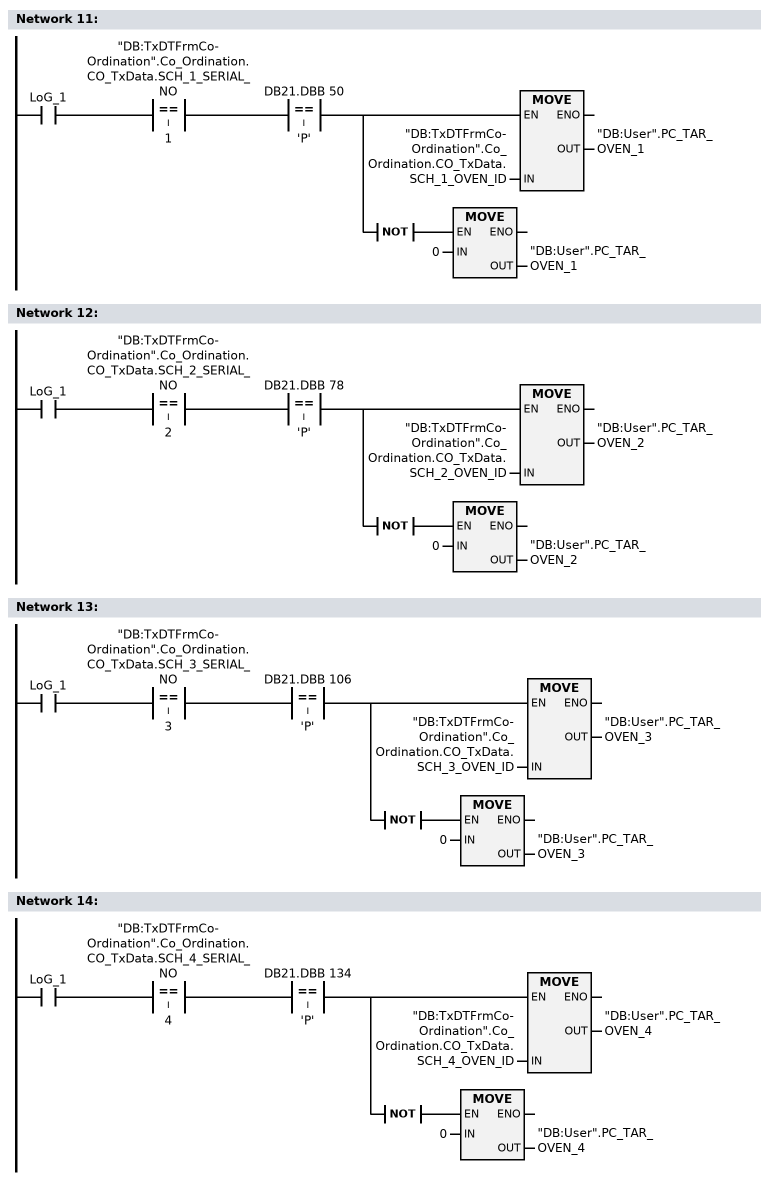
NETWORK
TITLE =
      A     "LoG_1";
      A(;
      L     "DB:TxDTFrmCo-Ordination".Co_Ordination.CO_TxData.SCH_1_SERIAL_NO;
      L     1;
      ==I;
      );
      A(;
      L     DB21.DBB 50;
      L     'P';
      ==I;
      );
      =     L 20.0;
      A     L 20.0;
      JNB   _01A;
      L     "DB:TxDTFrmCo-Ordination".Co_Ordination.CO_TxData.SCH_1_OVEN_ID;
      T     "DB:User".PC_TAR_OVEN_1;
_01A: NOP   0;
      A     L 20.0;
      NOT;
      JNB   _01B;
      L     0;
      T     "DB:User".PC_TAR_OVEN_1;
_01B: NOP   0;
NETWORK
TITLE =
      A     "LoG_1";
      A(;
      L     "DB:TxDTFrmCo-Ordination".Co_Ordination.CO_TxData.SCH_2_SERIAL_NO;
      L     2;
      ==I;
      );
      A(;
      L     DB21.DBB 78;
      L     'P';
      ==I;
      );
      =     L 21.0;
      A     L 21.0;
      JNB   _01C;
      L     "DB:TxDTFrmCo-Ordination".Co_Ordination.CO_TxData.SCH_2_OVEN_ID;
      T     "DB:User".PC_TAR_OVEN_2;
_01C: NOP   0;
      A     L 21.0;
      NOT;
      JNB   _01D;
      L     0;
      T     "DB:User".PC_TAR_OVEN_2;
_01D: NOP   0;
NETWORK
TITLE =
      A     "LoG_1";
      A(;
      L     "DB:TxDTFrmCo-Ordination".Co_Ordination.CO_TxData.SCH_3_SERIAL_NO;
      L     3;
      ==I;
      );
      A(;
      L     DB21.DBB 106;
      L     'P';
      ==I;
      );
      =     L 27.0;
      A     L 27.0;
      JNB   _01c;
      L     "DB:TxDTFrmCo-Ordination".Co_Ordination.CO_TxData.SCH_3_OVEN_ID;
      T     "DB:User".PC_TAR_OVEN_3;
_01c: NOP   0;
      A     L 27.0;
      NOT;
      JNB   _01d;
      L     0;
      T     "DB:User".PC_TAR_OVEN_3;
_01d: NOP   0;
NETWORK
TITLE =
      A     "LoG_1";
      A(;
      L     "DB:TxDTFrmCo-Ordination".Co_Ordination.CO_TxData.SCH_4_SERIAL_NO;
      L     4;
      ==I;
      );
      A(;
      L     DB21.DBB 134;
      L     'P';
      ==I;
      );
      =     L 28.0;
      A     L 28.0;
      JNB   _028;
      L     "DB:TxDTFrmCo-Ordination".Co_Ordination.CO_TxData.SCH_4_OVEN_ID;
      T     "DB:User".PC_TAR_OVEN_4;
_028: NOP   0;
      A     L 28.0;
      NOT;
      JNB   _029;
      L     0;
      T     "DB:User".PC_TAR_OVEN_4;
_029: NOP   0;
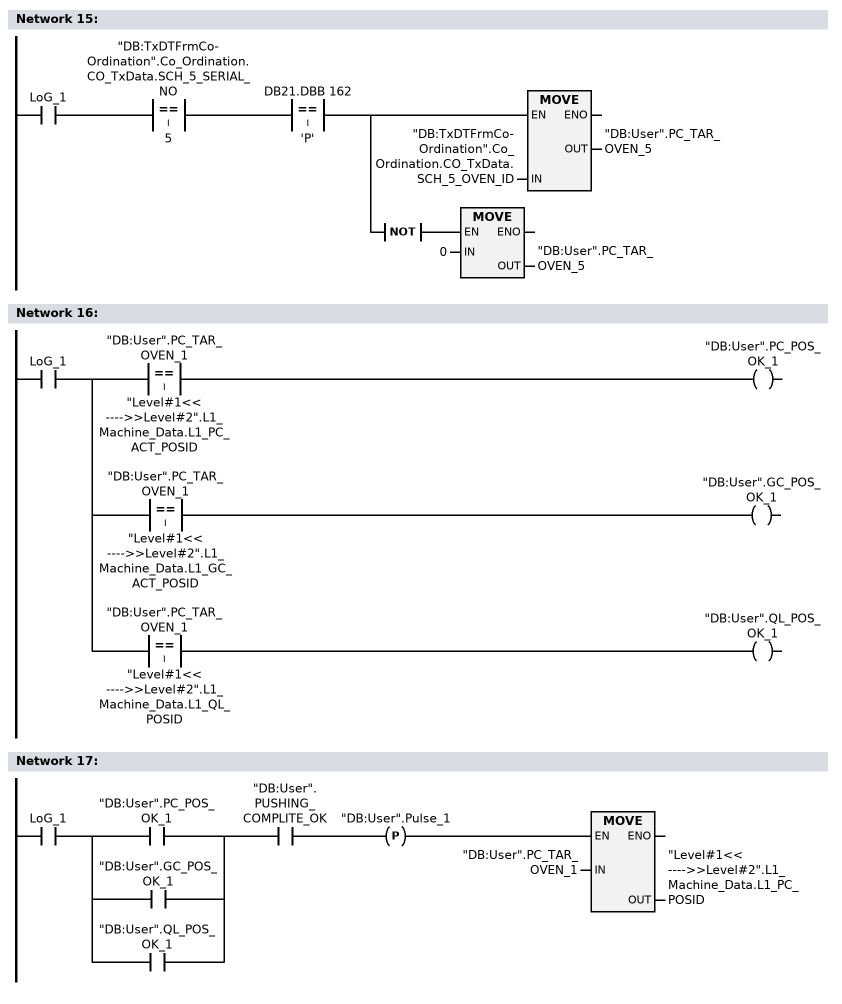
NETWORK
TITLE =
      A     "LoG_1";
      A(;
      L     "DB:TxDTFrmCo-Ordination".Co_Ordination.CO_TxData.SCH_5_SERIAL_NO;
      L     5;
      ==I;
      );
      A(;
      L     DB21.DBB 162;
      L     'P';
      ==I;
      );
      =     L 29.0;
      A     L 29.0;
      JNB   _02a;
      L     "DB:TxDTFrmCo-Ordination".Co_Ordination.CO_TxData.SCH_5_OVEN_ID;
      T     "DB:User".PC_TAR_OVEN_5;
_02a: NOP   0;
      A     L 29.0;
      NOT;
      JNB   _02b;
      L     0;
      T     "DB:User".PC_TAR_OVEN_5;
_02b: NOP   0;
NETWORK
TITLE =
      A     "LoG_1";
      =     L 30.0;
      A     L 30.0;
      A(;
      L     "DB:User".PC_TAR_OVEN_1;
      L     "Level#1<< ---->>Level#2".L1_Machine_Data.L1_PC_ACT_POSID;
      ==I;
      );
      =     "DB:User".PC_POS_OK_1;
      A     L 30.0;
      A(;
      L     "DB:User".PC_TAR_OVEN_1;
      L     "Level#1<< ---->>Level#2".L1_Machine_Data.L1_GC_ACT_POSID;
      ==I;
      );
      =     "DB:User".GC_POS_OK_1;
      A     L 30.0;
      A(;
      L     "DB:User".PC_TAR_OVEN_1;
      L     "Level#1<< ---->>Level#2".L1_Machine_Data.L1_QL_POSID;
      ==I;
      );
      =     "DB:User".QL_POS_OK_1;
NETWORK
TITLE =
      A     "LoG_1";
      A(;
      O     "DB:User".PC_POS_OK_1;
      O     "DB:User".GC_POS_OK_1;
      O     "DB:User".QL_POS_OK_1;
      );
      A     "DB:User".PUSHING_COMPLITE_OK;
      FP    "DB:User".Pulse_1;
      JNB   _022;
      L     "DB:User".PC_TAR_OVEN_1;
      T     "Level#1<< ---->>Level#2".L1_Machine_Data.L1_PC_POSID;
_022: NOP   0;
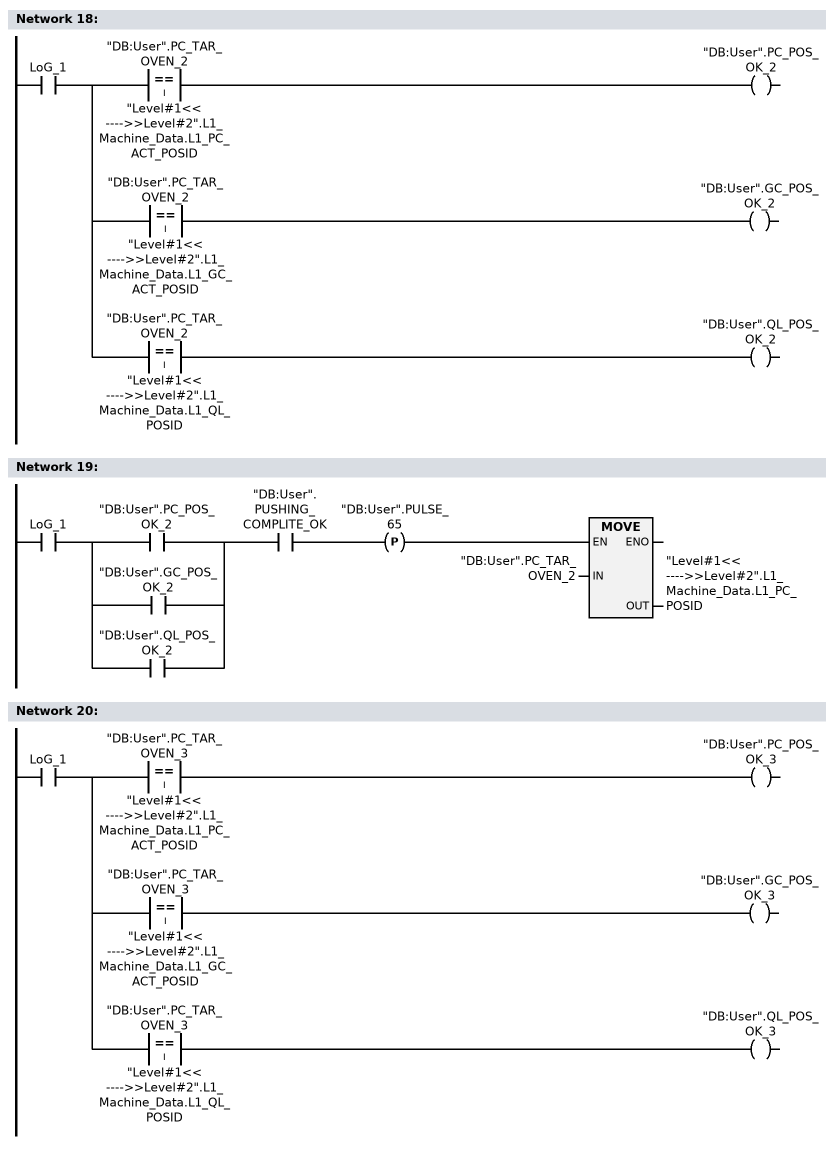
NETWORK
TITLE =
      A     "LoG_1";
      =     L 30.0;
      A     L 30.0;
      A(;
      L     "DB:User".PC_TAR_OVEN_2;
      L     "Level#1<< ---->>Level#2".L1_Machine_Data.L1_PC_ACT_POSID;
      ==I;
      );
      =     "DB:User".PC_POS_OK_2;
      A     L 30.0;
      A(;
      L     "DB:User".PC_TAR_OVEN_2;
      L     "Level#1<< ---->>Level#2".L1_Machine_Data.L1_GC_ACT_POSID;
      ==I;
      );
      =     "DB:User".GC_POS_OK_2;
      A     L 30.0;
      A(;
      L     "DB:User".PC_TAR_OVEN_2;
      L     "Level#1<< ---->>Level#2".L1_Machine_Data.L1_QL_POSID;
      ==I;
      );
      =     "DB:User".QL_POS_OK_2;
NETWORK
TITLE =
      A     "LoG_1";
      A(;
      O     "DB:User".PC_POS_OK_2;
      O     "DB:User".GC_POS_OK_2;
      O     "DB:User".QL_POS_OK_2;
      );
      A     "DB:User".PUSHING_COMPLITE_OK;
      FP    "DB:User".PULSE_65;
      JNB   _023;
      L     "DB:User".PC_TAR_OVEN_2;
      T     "Level#1<< ---->>Level#2".L1_Machine_Data.L1_PC_POSID;
_023: NOP   0;
NETWORK
TITLE =
      A     "LoG_1";
      =     L 30.0;
      A     L 30.0;
      A(;
      L     "DB:User".PC_TAR_OVEN_3;
      L     "Level#1<< ---->>Level#2".L1_Machine_Data.L1_PC_ACT_POSID;
      ==I;
      );
      =     "DB:User".PC_POS_OK_3;
      A     L 30.0;
      A(;
      L     "DB:User".PC_TAR_OVEN_3;
      L     "Level#1<< ---->>Level#2".L1_Machine_Data.L1_GC_ACT_POSID;
      ==I;
      );
      =     "DB:User".GC_POS_OK_3;
      A     L 30.0;
      A(;
      L     "DB:User".PC_TAR_OVEN_3;
      L     "Level#1<< ---->>Level#2".L1_Machine_Data.L1_QL_POSID;
      ==I;
      );
      =     "DB:User".QL_POS_OK_3;
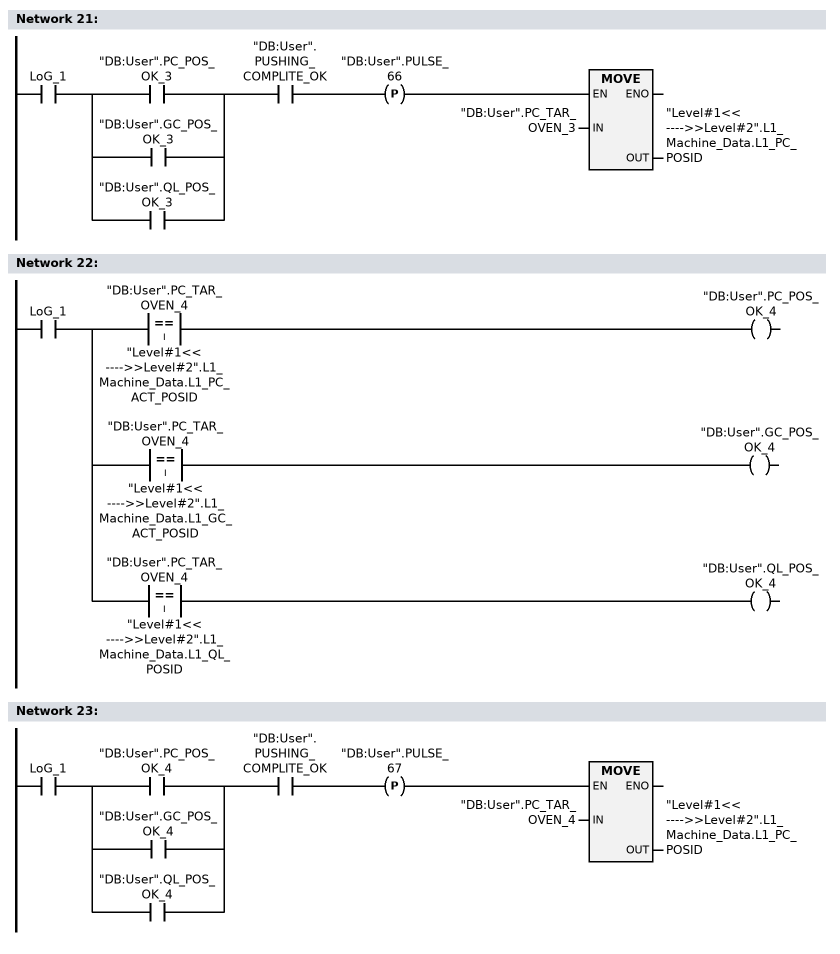
NETWORK
TITLE =
      A     "LoG_1";
      A(;
      O     "DB:User".PC_POS_OK_3;
      O     "DB:User".GC_POS_OK_3;
      O     "DB:User".QL_POS_OK_3;
      );
      A     "DB:User".PUSHING_COMPLITE_OK;
      FP    "DB:User".PULSE_66;
      JNB   _026;
      L     "DB:User".PC_TAR_OVEN_3;
      T     "Level#1<< ---->>Level#2".L1_Machine_Data.L1_PC_POSID;
_026: NOP   0;
NETWORK
TITLE =
      A     "LoG_1";
      =     L 30.0;
      A     L 30.0;
      A(;
      L     "DB:User".PC_TAR_OVEN_4;
      L     "Level#1<< ---->>Level#2".L1_Machine_Data.L1_PC_ACT_POSID;
      ==I;
      );
      =     "DB:User".PC_POS_OK_4;
      A     L 30.0;
      A(;
      L     "DB:User".PC_TAR_OVEN_4;
      L     "Level#1<< ---->>Level#2".L1_Machine_Data.L1_GC_ACT_POSID;
      ==I;
      );
      =     "DB:User".GC_POS_OK_4;
      A     L 30.0;
      A(;
      L     "DB:User".PC_TAR_OVEN_4;
      L     "Level#1<< ---->>Level#2".L1_Machine_Data.L1_QL_POSID;
      ==I;
      );
      =     "DB:User".QL_POS_OK_4;
NETWORK
TITLE =
      A     "LoG_1";
      A(;
      O     "DB:User".PC_POS_OK_4;
      O     "DB:User".GC_POS_OK_4;
      O     "DB:User".QL_POS_OK_4;
      );
      A     "DB:User".PUSHING_COMPLITE_OK;
      FP    "DB:User".PULSE_67;
      JNB   _027;
      L     "DB:User".PC_TAR_OVEN_4;
      T     "Level#1<< ---->>Level#2".L1_Machine_Data.L1_PC_POSID;
_027: NOP   0;
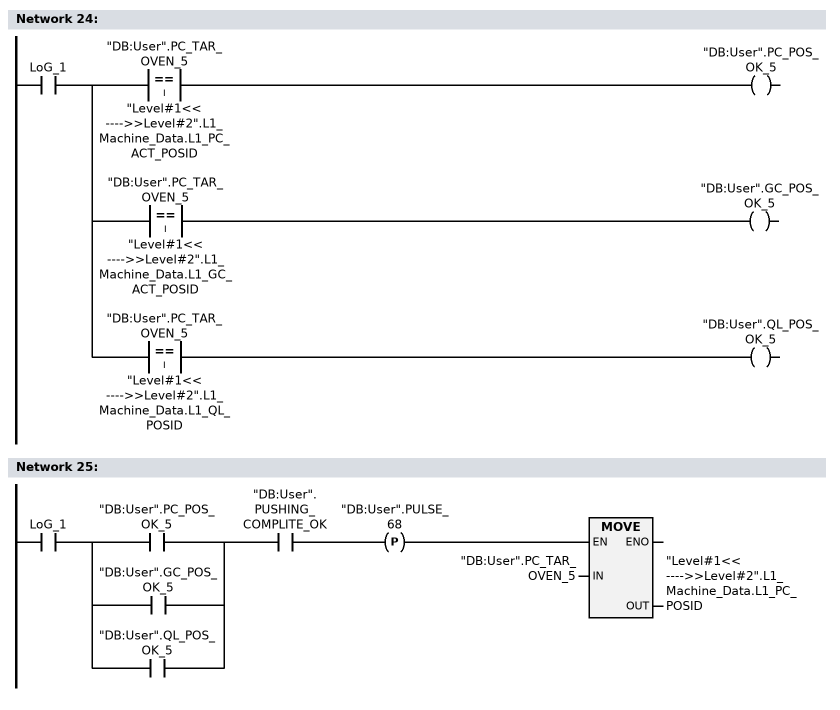
NETWORK
TITLE =
      A     "LoG_1";
      =     L 30.0;
      A     L 30.0;
      A(;
      L     "DB:User".PC_TAR_OVEN_5;
      L     "Level#1<< ---->>Level#2".L1_Machine_Data.L1_PC_ACT_POSID;
      ==I;
      );
      =     "DB:User".PC_POS_OK_5;
      A     L 30.0;
      A(;
      L     "DB:User".PC_TAR_OVEN_5;
      L     "Level#1<< ---->>Level#2".L1_Machine_Data.L1_GC_ACT_POSID;
      ==I;
      );
      =     "DB:User".GC_POS_OK_5;
      A     L 30.0;
      A(;
      L     "DB:User".PC_TAR_OVEN_5;
      L     "Level#1<< ---->>Level#2".L1_Machine_Data.L1_QL_POSID;
      ==I;
      );
      =     "DB:User".QL_POS_OK_5;
NETWORK
TITLE =
      A     "LoG_1";
      A(;
      O     "DB:User".PC_POS_OK_5;
      O     "DB:User".GC_POS_OK_5;
      O     "DB:User".QL_POS_OK_5;
      );
      A     "DB:User".PUSHING_COMPLITE_OK;
      FP    "DB:User".PULSE_68;
      JNB   _02c;
      L     "DB:User".PC_TAR_OVEN_5;
      T     "Level#1<< ---->>Level#2".L1_Machine_Data.L1_PC_POSID;
_02c: NOP   0;
NETWORK
TITLE =
END_FUNCTION

FUNCTION "FC:CoPLC-------->HMI" : VOID	// FC 26
VERSION : 0.1
BEGIN
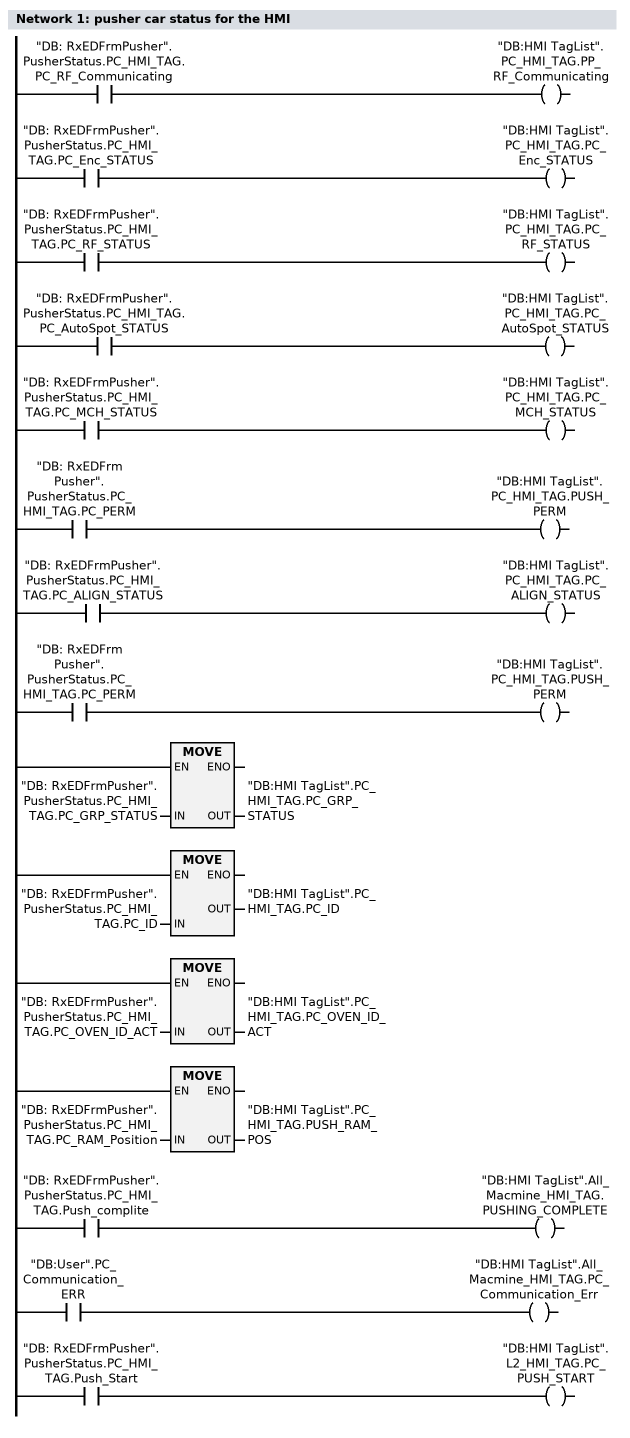
NETWORK
TITLE = pusher car status for the HMI
      A     "DB: RxEDFrmPusher".PusherStatus.PC_HMI_TAG.PC_RF_Communicating;
      =     "DB:HMI TagList".PC_HMI_TAG.PP_RF_Communicating;
//..
      A     "DB: RxEDFrmPusher".PusherStatus.PC_HMI_TAG.PC_Enc_STATUS;
      =     "DB:HMI TagList".PC_HMI_TAG.PC_Enc_STATUS;
//..
      A     "DB: RxEDFrmPusher".PusherStatus.PC_HMI_TAG.PC_RF_STATUS;
      =     "DB:HMI TagList".PC_HMI_TAG.PC_RF_STATUS;
//..
      A     "DB: RxEDFrmPusher".PusherStatus.PC_HMI_TAG.PC_AutoSpot_STATUS;
      =     "DB:HMI TagList".PC_HMI_TAG.PC_AutoSpot_STATUS;
//..
      A     "DB: RxEDFrmPusher".PusherStatus.PC_HMI_TAG.PC_MCH_STATUS;
      =     "DB:HMI TagList".PC_HMI_TAG.PC_MCH_STATUS;
//..
      A     "DB: RxEDFrmPusher".PusherStatus.PC_HMI_TAG.PC_PERM;
      =     "DB:HMI TagList".PC_HMI_TAG.PUSH_PERM;
//..
      A     "DB: RxEDFrmPusher".PusherStatus.PC_HMI_TAG.PC_ALIGN_STATUS;
      =     "DB:HMI TagList".PC_HMI_TAG.PC_ALIGN_STATUS;
//..
      A     "DB: RxEDFrmPusher".PusherStatus.PC_HMI_TAG.PC_PERM;
      =     "DB:HMI TagList".PC_HMI_TAG.PUSH_PERM;
//..
      L     "DB: RxEDFrmPusher".PusherStatus.PC_HMI_TAG.PC_GRP_STATUS;
      T     "DB:HMI TagList".PC_HMI_TAG.PC_GRP_STATUS;
//..
      L     "DB: RxEDFrmPusher".PusherStatus.PC_HMI_TAG.PC_ID;
      T     "DB:HMI TagList".PC_HMI_TAG.PC_ID;
//..
      L     "DB: RxEDFrmPusher".PusherStatus.PC_HMI_TAG.PC_OVEN_ID_ACT;
      T     "DB:HMI TagList".PC_HMI_TAG.PC_OVEN_ID_ACT;
//..
      L     "DB: RxEDFrmPusher".PusherStatus.PC_HMI_TAG.PC_RAM_Position;
      T     "DB:HMI TagList".PC_HMI_TAG.PUSH_RAM_POS;
//..
      A     "DB: RxEDFrmPusher".PusherStatus.PC_HMI_TAG.Push_complite;
      =     "DB:HMI TagList".All_Macmine_HMI_TAG.PUSHING_COMPLETE;
//..
      A     "DB:User".PC_Communication_ERR;
      =     "DB:HMI TagList".All_Macmine_HMI_TAG.PC_Communication_Err;
//..
      A     "DB: RxEDFrmPusher".PusherStatus.PC_HMI_TAG.Push_Start;
      =     "DB:HMI TagList".L2_HMI_TAG.PC_PUSH_START;
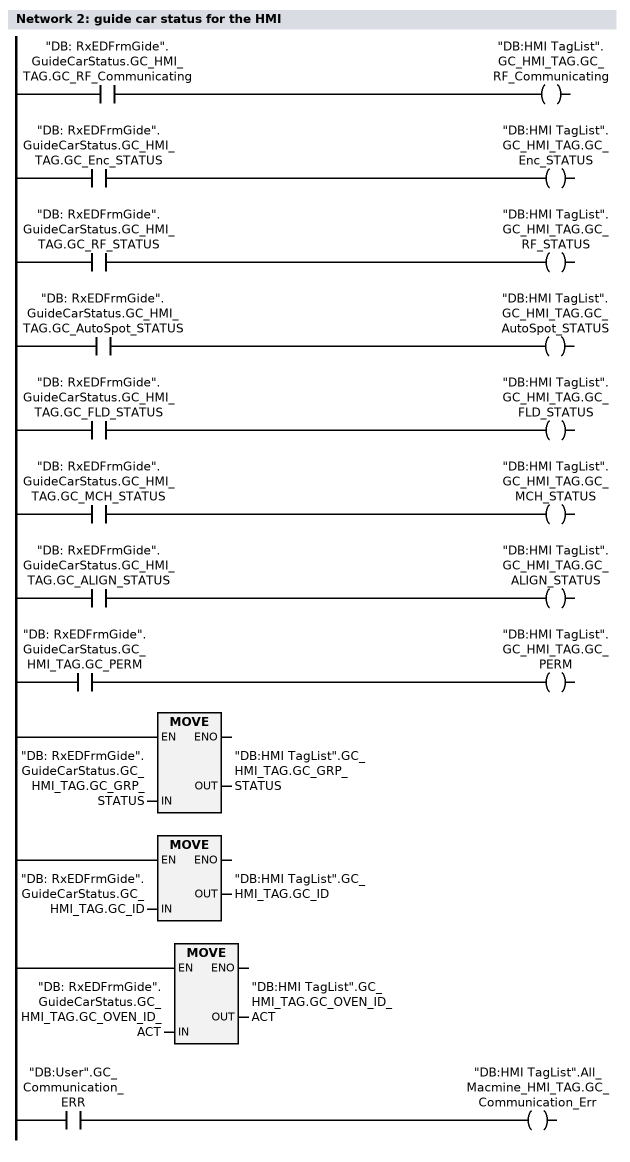
NETWORK
TITLE = guide car status for the HMI
      A     "DB: RxEDFrmGide".GuideCarStatus.GC_HMI_TAG.GC_RF_Communicating;
      =     "DB:HMI TagList".GC_HMI_TAG.GC_RF_Communicating;
//..
      A     "DB: RxEDFrmGide".GuideCarStatus.GC_HMI_TAG.GC_Enc_STATUS;
      =     "DB:HMI TagList".GC_HMI_TAG.GC_Enc_STATUS;
//..
      A     "DB: RxEDFrmGide".GuideCarStatus.GC_HMI_TAG.GC_RF_STATUS;
      =     "DB:HMI TagList".GC_HMI_TAG.GC_RF_STATUS;
//..
      A     "DB: RxEDFrmGide".GuideCarStatus.GC_HMI_TAG.GC_AutoSpot_STATUS;
      =     "DB:HMI TagList".GC_HMI_TAG.GC_AutoSpot_STATUS;
//..
      A     "DB: RxEDFrmGide".GuideCarStatus.GC_HMI_TAG.GC_FLD_STATUS;
      =     "DB:HMI TagList".GC_HMI_TAG.GC_FLD_STATUS;
//..
      A     "DB: RxEDFrmGide".GuideCarStatus.GC_HMI_TAG.GC_MCH_STATUS;
      =     "DB:HMI TagList".GC_HMI_TAG.GC_MCH_STATUS;
//..
      A     "DB: RxEDFrmGide".GuideCarStatus.GC_HMI_TAG.GC_ALIGN_STATUS;
      =     "DB:HMI TagList".GC_HMI_TAG.GC_ALIGN_STATUS;
//..
      A     "DB: RxEDFrmGide".GuideCarStatus.GC_HMI_TAG.GC_PERM;
      =     "DB:HMI TagList".GC_HMI_TAG.GC_PERM;
//..
      L     "DB: RxEDFrmGide".GuideCarStatus.GC_HMI_TAG.GC_GRP_STATUS;
      T     "DB:HMI TagList".GC_HMI_TAG.GC_GRP_STATUS;
//..
      L     "DB: RxEDFrmGide".GuideCarStatus.GC_HMI_TAG.GC_ID;
      T     "DB:HMI TagList".GC_HMI_TAG.GC_ID;
//..
      L     "DB: RxEDFrmGide".GuideCarStatus.GC_HMI_TAG.GC_OVEN_ID_ACT;
      T     "DB:HMI TagList".GC_HMI_TAG.GC_OVEN_ID_ACT;
//..
      A     "DB:User".GC_Communication_ERR;
      =     "DB:HMI TagList".All_Macmine_HMI_TAG.GC_Communication_Err;
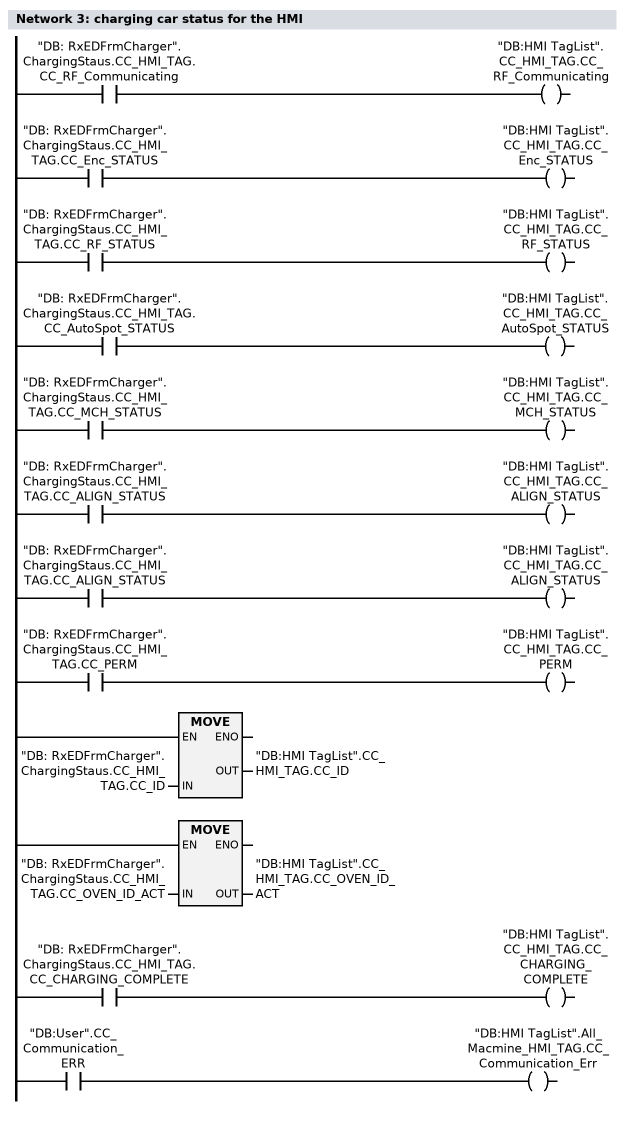
NETWORK
TITLE = charging car status for the HMI
      A     "DB: RxEDFrmCharger".ChargingStaus.CC_HMI_TAG.CC_RF_Communicating;
      =     "DB:HMI TagList".CC_HMI_TAG.CC_RF_Communicating;
//..
      A     "DB: RxEDFrmCharger".ChargingStaus.CC_HMI_TAG.CC_Enc_STATUS;
      =     "DB:HMI TagList".CC_HMI_TAG.CC_Enc_STATUS;
//..
      A     "DB: RxEDFrmCharger".ChargingStaus.CC_HMI_TAG.CC_RF_STATUS;
      =     "DB:HMI TagList".CC_HMI_TAG.CC_RF_STATUS;
//..
      A     "DB: RxEDFrmCharger".ChargingStaus.CC_HMI_TAG.CC_AutoSpot_STATUS;
      =     "DB:HMI TagList".CC_HMI_TAG.CC_AutoSpot_STATUS;
//..
      A     "DB: RxEDFrmCharger".ChargingStaus.CC_HMI_TAG.CC_MCH_STATUS;
      =     "DB:HMI TagList".CC_HMI_TAG.CC_MCH_STATUS;
//..
      A     "DB: RxEDFrmCharger".ChargingStaus.CC_HMI_TAG.CC_ALIGN_STATUS;
      =     "DB:HMI TagList".CC_HMI_TAG.CC_ALIGN_STATUS;
//..
      A     "DB: RxEDFrmCharger".ChargingStaus.CC_HMI_TAG.CC_ALIGN_STATUS;
      =     "DB:HMI TagList".CC_HMI_TAG.CC_ALIGN_STATUS;
//..
      A     "DB: RxEDFrmCharger".ChargingStaus.CC_HMI_TAG.CC_PERM;
      =     "DB:HMI TagList".CC_HMI_TAG.CC_PERM;
//..
      L     "DB: RxEDFrmCharger".ChargingStaus.CC_HMI_TAG.CC_ID;
      T     "DB:HMI TagList".CC_HMI_TAG.CC_ID;
//..
      L     "DB: RxEDFrmCharger".ChargingStaus.CC_HMI_TAG.CC_OVEN_ID_ACT;
      T     "DB:HMI TagList".CC_HMI_TAG.CC_OVEN_ID_ACT;
//..
      A     "DB: RxEDFrmCharger".ChargingStaus.CC_HMI_TAG.CC_CHARGING_COMPLETE;
      =     "DB:HMI TagList".CC_HMI_TAG.CC_CHARGING_COMPLETE;
//..
      A     "DB:User".CC_Communication_ERR;
      =     "DB:HMI TagList".All_Macmine_HMI_TAG.CC_Communication_Err;
//..
